FUNCTION_BLOCK "Banda_Poj_+Tryb_Reczny"	// FB 33
//Funkcja realizujaca koncepcje bandy pojedycznej, ktora uwzglednia rowniez tryb 
//reczny. W celu lepszego sterowania trybem recznym nalezy do³o¿yæ:
//-fotokomorki na tyle bandy.
//-fotokomorka na tyle okresla rowniez zajetosc
//-jazda do tylu bandy mozliwa
//-jazda do przodu poza fotokomorke mozliwa gdy nastepna w ruchu i wolna.
//-do³o¿enie okresnia trybu reczny/auto gdzie auto to 1 
//
AUTHOR : Kng
FAMILY : Bandy
NAME : B_dual
VERSION : 0.0
VAR_INPUT
  i_Marka_Bezpieczenstwa : BOOL ;
  i_Rezerwa_1 : BOOL ;	//Zamrozenie stanu pracy
  i_Auto_Reczny : BOOL ;	//1-auto,0-reczny
  i_Foto_Przod : BOOL ;	//Foto na koncu tasmy
  i_Foto_Tyl : BOOL ;	//Foto zapobiegajace wyjechaniu palety do tylu
  i_Zez_Od_Nast : BOOL ;
  i_Paleta_Dost_Od_Nast : BOOL ;
  i_Zez_Reczny_Od_Nast : BOOL ;
  i_Zabierz_Od_Pop : BOOL ;
  i_Zez_Reczny_Od_Pop : BOOL ;
  i_PB_Jazda_Tyl : BOOL ;
  i_PB_Jazda_Przod : BOOL ;
  Czas_Kontroli_Przejazdu : TIME ;
END_VAR
VAR_OUTPUT
  o_Zabierz_Do_Nast : BOOL ;	//Rozkaz pobrania do nast bandy
  o_Zez_Do_Pop : BOOL ;
  o_Paleta_Dost_Do_Pop : BOOL ;
  o_Motor_Lewo : BOOL ;
  o_Motor_Prawo : BOOL ;
  o_Zez_Reczny_Do_Nast : BOOL ;
  o_Zez_Reczny_Do_Pop : BOOL ;
  o_Zajetosc_Nieb : BOOL ;	//Dla bezpieczenstwa transportu
END_VAR
VAR
  Czas_kontrolny : FB 21;
  Help_A_Motor_Lewo : BOOL ;
  S_Help_Zab_Od_Pop : BOOL ;
  Stop_Czas_Kontrolny : BOOL ;
  Zbocze_1 : BOOL ;
  Zbocze_2 : BOOL ;
  Blokada_Wjazdu : BOOL ;
  Help_H_Motor_Prawo : BOOL ;
  Help_H_Motor_Lewo : BOOL ;
  Toggle : BOOL ;	//bit przemienny dla auto i hand
  Help_8 : BOOL ;
  Help_9 : BOOL ;
END_VAR
VAR_TEMP
  Temp_Help_1 : BOOL ;
  Temp_Help_2 : BOOL ;
  Czas_zadany : TIME ;
  Czas_aktualny : TIME ;
END_VAR
BEGIN
NETWORK
TITLE =
//
// B1        B2         foto_1    foto_2         B5        B6
//(\\\\\\\\\\\\\\\\\\)  (\\\\\\\\\\\\\\\\\\)  (\\\\\\\\\\\\\\\\\\)
//                  M1                    M2                     M3
//         
//        zabierz <-- pobierz      |  zabierz    <--  pobierz  
//     zez_do_pop --> zez_od_nast  |  zez_od_pop -->  zez_od_nast
//                                  
//-Uklad dzielony jest na realizowane funkcje
//
//         <----------------------------------------- kierunek
//                  
//
// ten network celowo jest pusty
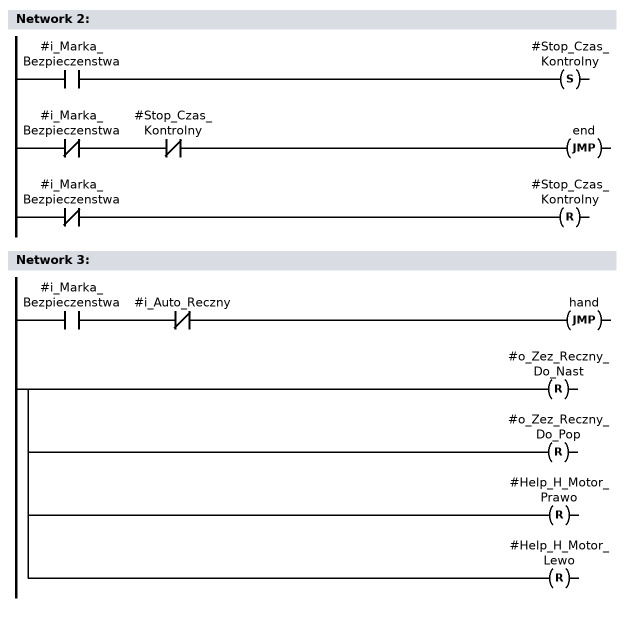
NETWORK
TITLE =
//Sprawdzenie stanu bezpieczenstwa lub freeze
//Skocz jezeli brak marki bezpieczenstwa
//Marka bezpieczenstwa ok gdy wysoki
      A     #i_Marka_Bezpieczenstwa;
      S     #Stop_Czas_Kontrolny;
      AN    #i_Marka_Bezpieczenstwa;
      AN    #Stop_Czas_Kontrolny;
      JC    end;
      AN    #i_Marka_Bezpieczenstwa;
      R     #Stop_Czas_Kontrolny;
NETWORK
TITLE =
//Wyznczenie zbocza pozytywnego i negatywnego
//skok do trybu recznego 
      A     #i_Marka_Bezpieczenstwa;
      AN    #i_Auto_Reczny;
      JC    hand;
//czyszczenie trybu recznego
      SET;
      R     #o_Zez_Reczny_Do_Nast;
      R     #o_Zez_Reczny_Do_Pop;
      R     #Help_H_Motor_Prawo;
      R     #Help_H_Motor_Lewo;
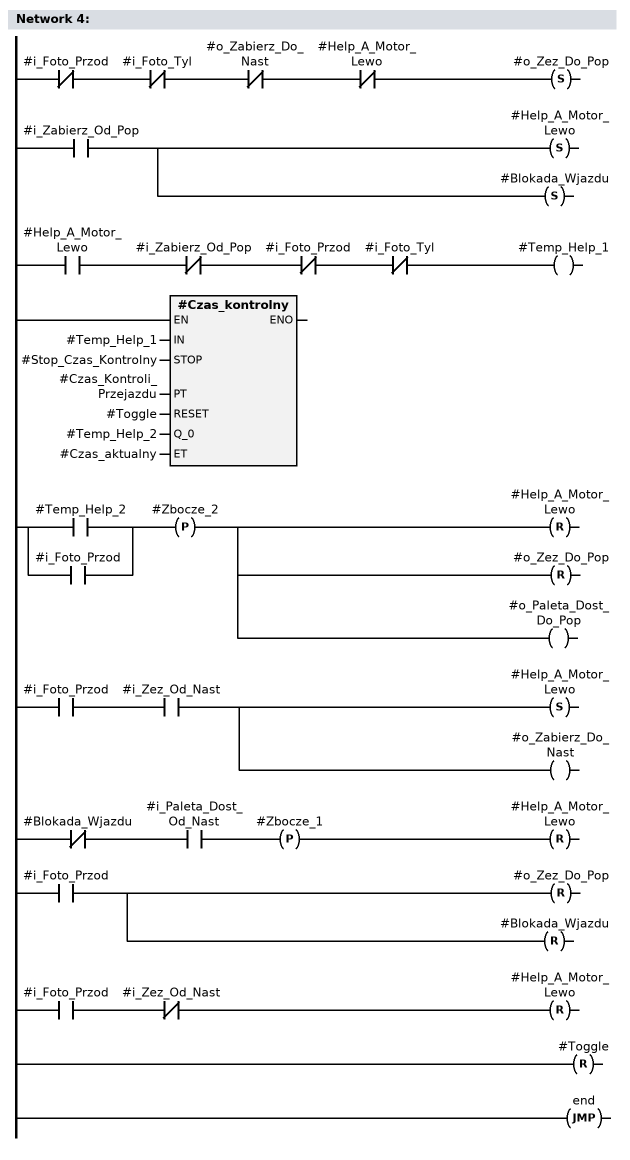
NETWORK
TITLE =
// Opis poszczegolnych krokow i skok do nich
// Tasma poprzednia pusta i bierzaca pusta
      AN    #i_Foto_Przod;
      AN    #i_Foto_Tyl;	//dodano bo hand
      AN    #o_Zabierz_Do_Nast;
      AN    #Help_A_Motor_Lewo;
      S     #o_Zez_Do_Pop;
      A     #i_Zabierz_Od_Pop;
      S     #Help_A_Motor_Lewo;
      S     #Blokada_Wjazdu;
//Warunek gdy pobranie z poprzedniej i miejsce foto srodek
//jest zajete
      A     #Help_A_Motor_Lewo;
      AN    #i_Zabierz_Od_Pop;
      AN    #i_Foto_Przod;
      AN    #i_Foto_Tyl;	//dodano bo hand
      =     #Temp_Help_1;
      CALL  #Czas_kontrolny (
           IN                       := #Temp_Help_1,
           STOP                     := #Stop_Czas_Kontrolny,
           PT                       := #Czas_Kontroli_Przejazdu,
           RESET                    := #Toggle,
           Q_0                      := #Temp_Help_2,
           ET                       := #Czas_aktualny);
//Paleta dostarczona
      A     #Temp_Help_2;
      O;
      A     #i_Foto_Przod;
      FP    #Zbocze_2;
      R     #Help_A_Motor_Lewo;
      R     #o_Zez_Do_Pop;
      =     #o_Paleta_Dost_Do_Pop;
//jest zezwolenie od nastepnej
      A     #i_Foto_Przod;
      A     #i_Zez_Od_Nast;
      S     #Help_A_Motor_Lewo;
      =     #o_Zabierz_Do_Nast;
//Potwierdzenie otrzymania palety
      AN    #Blokada_Wjazdu;
      A     #i_Paleta_Dost_Od_Nast;
      FP    #Zbocze_1;
      R     #Help_A_Motor_Lewo;
//Gdy zajete Foto_1 brak zezwolenia do poprzedniej
      A     #i_Foto_Przod;
      R     #o_Zez_Do_Pop;
      R     #Blokada_Wjazdu;
//warunkowe zakonczenie pracy silnika gdy brak zezwolenia
//z nastepnej
      A     #i_Foto_Przod;
      AN    #i_Zez_Od_Nast;
      R     #Help_A_Motor_Lewo;
//wylacz toggle
      SET;
      R     #Toggle;
//skocz do koniec
      JU    end;
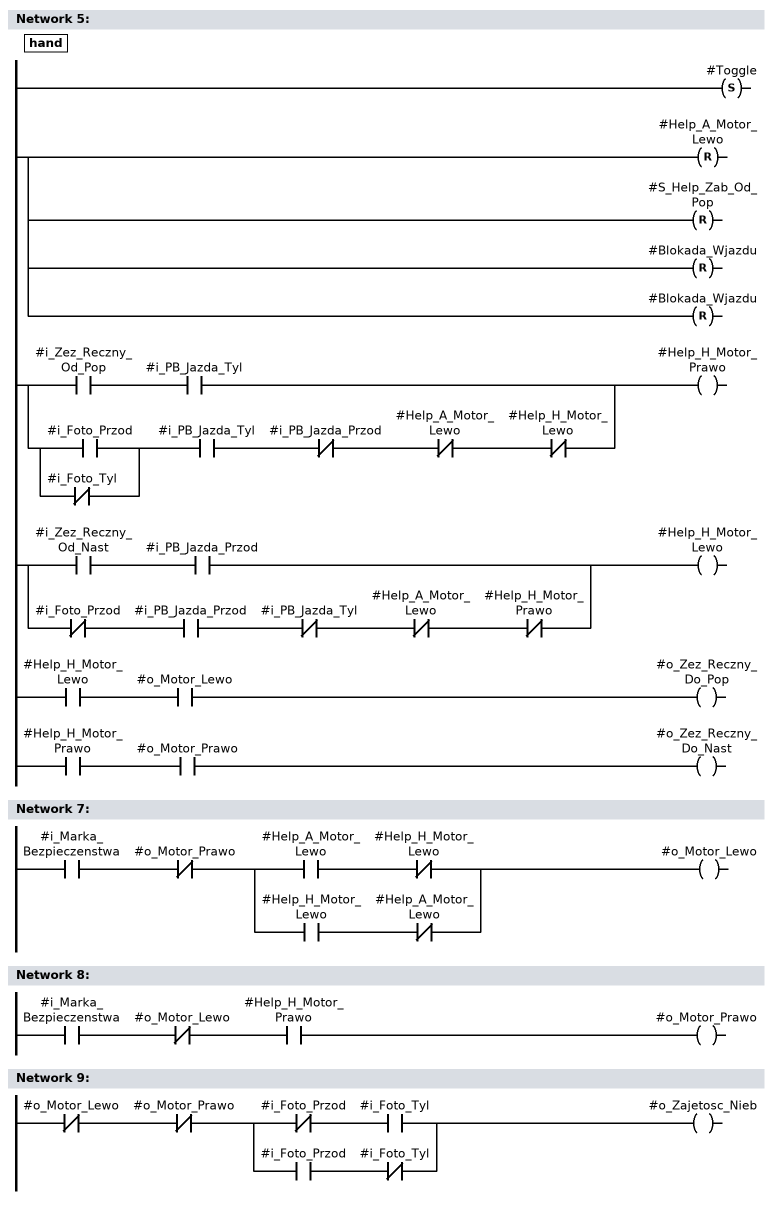
NETWORK
TITLE =
//Tryb reczny
//
hand: NOP   0;
//wlacz toggle
      SET;
      S     #Toggle;
//czyszczenie bitow z automatyki
      SET;
      R     #Help_A_Motor_Lewo;
      R     #S_Help_Zab_Od_Pop;
      R     #Blokada_Wjazdu;
      R     #Blokada_Wjazdu;
//ustawienie przyciskow
//jazda do tylu przycisk tyl
      A     #i_Zez_Reczny_Od_Pop;
      A     #i_PB_Jazda_Tyl;
      O;
      A(;
      O     #i_Foto_Przod;
      ON    #i_Foto_Tyl;
      );
      A(;
      A     #i_PB_Jazda_Tyl;
      AN    #i_PB_Jazda_Przod;
      AN    #Help_A_Motor_Lewo;
      AN    #Help_H_Motor_Lewo;
      );
      =     #Help_H_Motor_Prawo;
//jazda do przodu
      A     #i_Zez_Reczny_Od_Nast;
      A     #i_PB_Jazda_Przod;
      O;
      AN    #i_Foto_Przod;
      A(;
      A     #i_PB_Jazda_Przod;
      AN    #i_PB_Jazda_Tyl;
      AN    #Help_A_Motor_Lewo;
      AN    #Help_H_Motor_Prawo;
      );
      =     #Help_H_Motor_Lewo;
//wystawienie zezwolen do innych band wspolpracujacych recznie
//zezwolenie do tylu 
//zezwolenie do poprzedniej
      A     #Help_H_Motor_Lewo;
      A     #o_Motor_Lewo;
      =     #o_Zez_Reczny_Do_Pop;
//zezwolenie do nastepnej
      A     #Help_H_Motor_Prawo;
      A     #o_Motor_Prawo;
      =     #o_Zez_Reczny_Do_Nast;
NETWORK
TITLE =
//Przypisanie wyjsc
//Koniec skoku
end:  NOP   0;
NETWORK
TITLE =
////jazda automatyka reczny przod
      A     #i_Marka_Bezpieczenstwa;
      AN    #o_Motor_Prawo;
      A(;
      A     #Help_A_Motor_Lewo;
      AN    #Help_H_Motor_Lewo;
      O;
      A     #Help_H_Motor_Lewo;
      AN    #Help_A_Motor_Lewo;
      );
      =     #o_Motor_Lewo;
NETWORK
TITLE =
////Jazda reczny tyl
      A     #i_Marka_Bezpieczenstwa;
      AN    #o_Motor_Lewo;
      A     #Help_H_Motor_Prawo;
      =     #o_Motor_Prawo;
NETWORK
TITLE =
//Zajetosc
      AN    #o_Motor_Lewo;
      AN    #o_Motor_Prawo;
      A(;
      AN    #i_Foto_Przod;
      A     #i_Foto_Tyl;
      O;
      A     #i_Foto_Przod;
      AN    #i_Foto_Tyl;
      );
      =     #o_Zajetosc_Nieb;
NETWORK
TITLE =
//Koniec
//koniec
      BEU;
END_FUNCTION_BLOCK

FUNCTION_BLOCK "Banda_Obr_Bind"	// FB 34
//Program odpowiadajacy za bindowanie produktu na obrotnicy
//
//
AUTHOR : Kng
FAMILY : Bandy
NAME : Band_obr
VERSION : 0.1
VAR_INPUT
  i_Marka_Bezpieczenstwa : BOOL ;
  i_Auto_Reczny : BOOL ;	//gdzie 1-Auto 0 Reczny
  i_Bindownica_Auto : BOOL ;	//Mro¿enie stanu pracy
  i_Foto_Tyl : BOOL ;	//foto poczatek
  i_Foto_Przod : BOOL ;	//foto koniec
  i_Zez_od_Nast : BOOL ;
  i_Zabierz_od_Pop : BOOL ;
  i_Paleta_Dost_Od_Nast : BOOL ;
  i_czuj_0_st_1 : BOOL ;	//0 stopni Wlot/Wylot
  i_czuj_0_st_2 : BOOL ;	//Hamowanie 0 stopni
  i_czuj_90_st_1 : BOOL ;	//Hamowanie 90 stopni
  i_czuj_90_st_2 : BOOL ;	//90 stopni
  i_Czuj_180_st_1 : BOOL ;	//Hamowanie 180 stopni
  i_Czuj_180_st_2 : BOOL ;	//180 stopni
  i_Czuj_270_st_1 : BOOL ;	//Hamowanie 270 stopni
  i_Czuj_270_st_2 : BOOL ;
  i_Bind_Obwod_Ok : BOOL ;	//270 stopni
  i_Bind_Poz_Podst : BOOL ;
  i_Bind_Syg_Got : BOOL ;
  i_Bind_Blad : BOOL ;
  i_Bind_Start_Kon : BOOL ;	//Bindownica start koniec wiazania
  i_PB_Obr_Prawo : BOOL ;
  i_PB_Obr_Lewo : BOOL ;
  i_Zawsze_True : BOOL ;	//Zawsze jeden do pomocy
  i_PB_Jazda_Przod : BOOL ;
  i_PB_Jazda_Tyl : BOOL ;
  i_PB_Cykl_Start : BOOL ;
  i_PB_Cykl_Stop : BOOL ;
  i_Zez_Reczny_Od_Pop : BOOL ;
  i_Zez_Reczny_Od_Nast : BOOL ;
  i_Reset_Krokow : BOOL ;
  i_Reset_Bledow : BOOL ;
  i_Rezerwa_1 : BOOL ;
  i_Rezerwa_2 : BOOL ;
  i_Rezerwa_3 : BOOL ;
  i_Rezerwa_4 : BOOL ;
END_VAR
VAR_OUTPUT
  o_Zez_do_Pop : BOOL ;
  o_Paleta_Dost_Do_Pop : BOOL ;
  o_Zabierz_do_Nast : BOOL ;
  o_Motor_1_lewo : BOOL ;
  o_Motor_1_prawo : BOOL ;
  o_Motor_1_Wolno : BOOL ;
  o_Motor_2_obr_s_Lewo : BOOL ;	//Motor obrotnicy,kierunek strona wejscia,szybko
  o_Motor_2_obr_s_Prawo : BOOL ;	//Motor obrotnicy,kierunek strona wyjscia,szybko
  o_Motor_2_Wolno : BOOL ;	//Motor obrotnicy,kierunek strona wejscia,wolno
  o_Bind_Zez_Na_Prace : BOOL ;
  o_Bind_Start_Wiazania : BOOL ;
  o_Bind_Blad_Ogolny : BOOL ;
  o_Zez_Reczny_do_Pop : BOOL ;
  o_Zez_Reczny_do_nast : BOOL ;
  o_Lampka_Bindowanie : BOOL ;
  o_Lampka_Przycisk_Reset : BOOL ;
  o_Blad_Cyklu : BOOL ;
  o_Blad_Ogolny : BOOL ;
  o_Cykl_Bindowania_Trwa : BOOL ;
  o_Rezerwa_2 : BOOL ;
  o_Rezerwa_3 : BOOL ;
END_VAR
VAR
  Sterowanie_Obrotu : FB 54;
  Pozycj_Obr : FB 55;
  Bindowanie : FB 35;
  Pozycjonowanie_Palety : FB 58;
  Kontrola_Rolki_Wlot : FB 20;
  Dojazd_Rolki_Wlot : FB 20;
  Opuszczenie_Bandy : FB 20;	//Czas kontrolny wjazdu palety
  Tim_Rezerwa_1 : FB 20;
  Tim_Rezerwa_2 : FB 20;
  Tim_Rezerwa_3 : SFB 4;	//Timer opozniajacy bindowanie
  Silniki_nie_pracuja : BOOL ;
  Help_A_Motor_1_lewo : BOOL ;
  Help_A_Motor_1_prawo : BOOL ;
  Help_A_Motor_1_wolno : BOOL ;
  Help_H_Motor_1_lewo : BOOL ;
  Help_H_Motor_1_prawo : BOOL ;
  Help_H_Motor_1_Wolno : BOOL ;
  Help_Motor_2_obr_lewo : BOOL ;
  Help_Motor_2_obr_prawo : BOOL ;
  Help_Motor_2_Wolno : BOOL ;
  Help_AP_Motor_1_Lewo : BOOL ;
  Help_AP_Motor_1_Prawo : BOOL ;
  Help_AP_Motor_1_Wolno : BOOL ;
  Pobranie_Wlot : BOOL ;
  Filtr_Rolki_Wlot : BOOL ;
  Stop_Czas_Kontrolny : BOOL ;
  H1_Doj_Rolki_Wlot : BOOL ;
  H2_Doj_Rolki_Wlot : BOOL ;
  Oddanie_Palety : BOOL ;
  Zbocze_1 : BOOL ;
  Toggle : BOOL ;	//Sygnal zamienny auto reczny
  Paleta_rowno_na_stan : BOOL ;
  Help_B_Zez_Na_Prace : BOOL ;
  Help_B_Start_Wiazan : BOOL ;
  Help_B_Blad_Ogolny : BOOL ;
  Help_Bin_Koniec_Cyklu : BOOL ;
  H_Start_Cyklu_Bind_Auto : BOOL ;
  H_Reset_Cyklu_Bind : BOOL ;
  H_Auto_Reczny : BOOL ;
  Auto_Reczny_W : BOOL ;
  Silnik_Rolek_Nie_Pracuje : BOOL ;
  Reset_Konca_Cyklu : BOOL ;
  Zbocze_2 : BOOL ;
  Help_PB_Start : BOOL ;
  H_Silnik_Rolek_Pracuje : BOOL ;
  H_Zez_do_Pop : BOOL ;
  H_Zabierz_do_Nast : BOOL ;
  H_Cykl_Bind_Trwa : BOOL ;
  Zbocze_3 : BOOL ;
  H_Blad_Cyklu : BOOL ;
  H_Marka_Bezp_Obr : BOOL ;
  H_Marka_Bezp_Poz : BOOL ;
  H_Auto_Reczny_Ster_Obr : BOOL ;
  H_Start_Cyklu_Bind_Recz : BOOL ;
  H_Reset_Srodka : BOOL ;	//Reset paleta na srodku
  H2_Start_Cyklu_Bind_Recz : BOOL ;
  H46 : BOOL ;
  H49 : BOOL ;
  H50 : BOOL ;
  Help_Cykl_Start_Reczny : BOOL ;
  H52 : BOOL ;
  H54 : BOOL ;
  H55 : BOOL ;
  H56 : BOOL ;
  H57 : BOOL ;
  H58 : INT ;
  H59 : BOOL ;
  H60 : BOOL ;	//Pozycja talerza osiagnieta
  H62 : BOOL ;
  H61 : INT ;
  H63 : BOOL ;
  H64 : BOOL ;
  H65 : BOOL ;
  H66 : BOOL ;
  H67 : BOOL ;
  H68 : BOOL ;
  H69 : BOOL ;
  H70 : BOOL ;
  H72 : BOOL ;
  H40 : BOOL ;
  H38 : BOOL ;
  H37 : BOOL ;
  H36 : BOOL ;
  H35 : BOOL ;
  H34 : BOOL ;
  H33 : BOOL ;
  H32 : BOOL ;
  H31 : BOOL ;
  H30 : BOOL ;
  H29 : BOOL ;
  H28 : BOOL ;	//Pozycjonowanie palety
  H27 : BOOL ;
  H26 : BOOL ;
END_VAR
VAR_TEMP
  Temp_Help_1 : BOOL ;
  Temp_Help_2 : BOOL ;
  Czas_zadany : TIME ;
  Czas_aktualny : TIME ;
  Czas_Kontroli_Przejazdu : TIME ;
  Czas_Monitora_Najazdu : TIME ;
  Czas_Opoznienia_Bind : TIME ;
END_VAR
BEGIN
NETWORK
TITLE =
//                   
//Wlot                                Wylot
//()()()()|()()()()|  ()()()  |()()()()|()()()()
//()()()()|()()()()| ()()()() |()()()()|()()()()
//()()()()|()()()()| ()()()() |()()()()|()()()()
//()()()()|()()()()| ()()()() |()()()()|()()()()
//()()()()|()()()()|  ()()()  |()()()()|()()()()
//
//      
//         
//          pobierz --> zabierz   |     pobierz --> zabierz   
//     zez_od_nast <-- zez_do_pop | zez_od_nast <-- zez_od_pop
//                                  
//-Uklad dzielony jest na realizowane funkcje
//
//         
//                  
//
// ten network celowo jest pusty
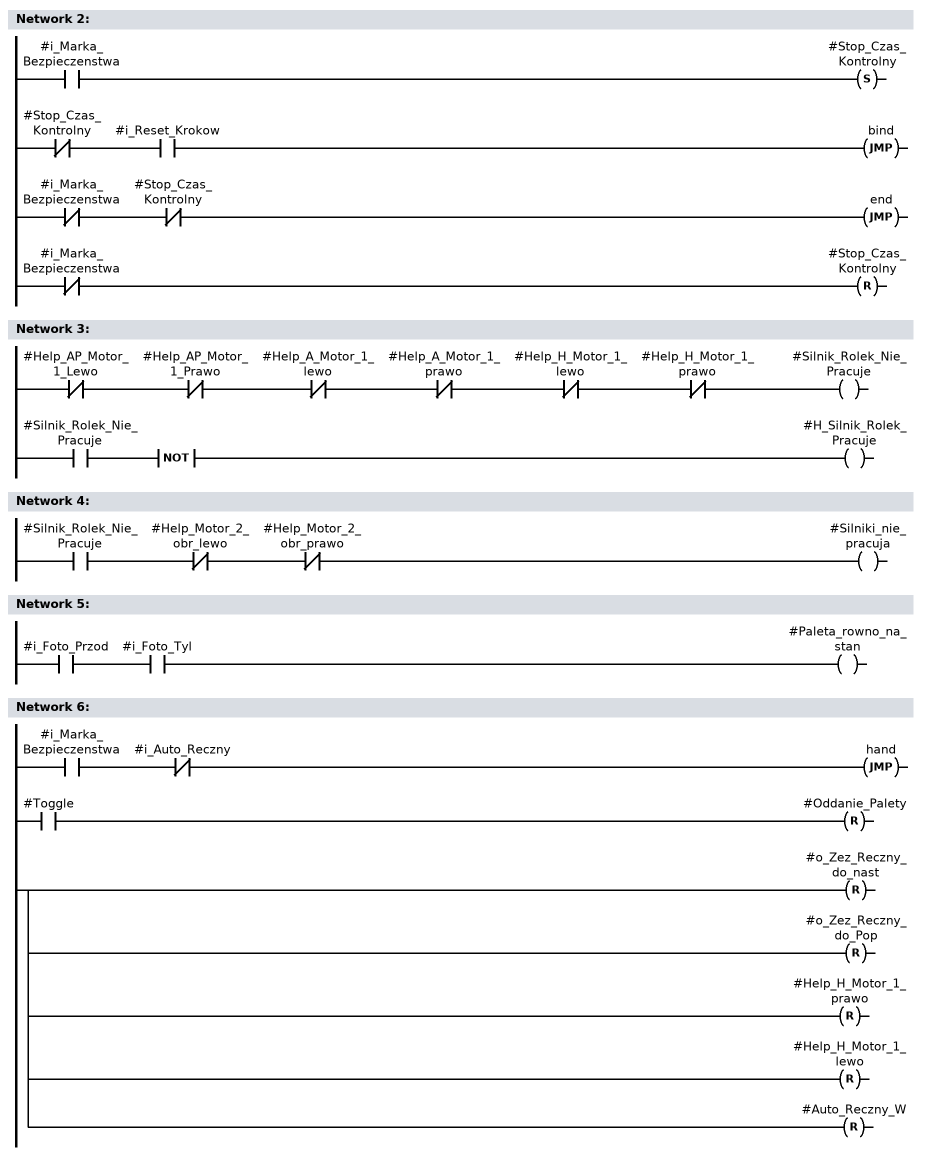
NETWORK
TITLE =
//Wyznczenie zbocza pozytywnego i negatywnego
//Skocz jezeli brak marki bezpieczenstwa
//Marka bezpieczenstwa ok gdy wysoki
//Freeze ok gdy niski
      A     #i_Marka_Bezpieczenstwa;
      S     #Stop_Czas_Kontrolny;
//skocz aby zrobic reset podczas stopu
      AN    #Stop_Czas_Kontrolny;
      A     #i_Reset_Krokow;
      JC    bind;
      AN    #i_Marka_Bezpieczenstwa;
      AN    #Stop_Czas_Kontrolny;
      JC    end;
      AN    #i_Marka_Bezpieczenstwa;
      R     #Stop_Czas_Kontrolny;
NETWORK
TITLE =
//Sprawdzenie czy rolki nie pracuja 
      AN    #Help_AP_Motor_1_Lewo;
      AN    #Help_AP_Motor_1_Prawo;
      AN    #Help_A_Motor_1_lewo;
      AN    #Help_A_Motor_1_prawo;
      AN    #Help_H_Motor_1_lewo;
      AN    #Help_H_Motor_1_prawo;
      =     #Silnik_Rolek_Nie_Pracuje;
      A     #Silnik_Rolek_Nie_Pracuje;
      NOT;
      =     #H_Silnik_Rolek_Pracuje;
NETWORK
TITLE =
//Silniki nie pracuja
//
      A     #Silnik_Rolek_Nie_Pracuje;
      AN    #Help_Motor_2_obr_lewo;
      AN    #Help_Motor_2_obr_prawo;
      =     #Silniki_nie_pracuja;
NETWORK
TITLE =
//Sprawdzenie czy paleta lezy na stanowisku
//sprawdzenie czy paleta lezy OK
      A     #i_Foto_Przod;
      A     #i_Foto_Tyl;
      =     #Paleta_rowno_na_stan;
NETWORK
TITLE =
//Skok do trybu recznego 
//skok do trybu recznego 
      A     #i_Marka_Bezpieczenstwa;
      AN    #i_Auto_Reczny;
      JC    hand;
//Powrot z trybu recznego do auto
      A     #Toggle;
      R     #Oddanie_Palety;
//czyszczenie trybu recznego
      SET;
      R     #o_Zez_Reczny_do_nast;
      R     #o_Zez_Reczny_do_Pop;
      R     #Help_H_Motor_1_prawo;
      R     #Help_H_Motor_1_lewo;
      R     #Auto_Reczny_W;
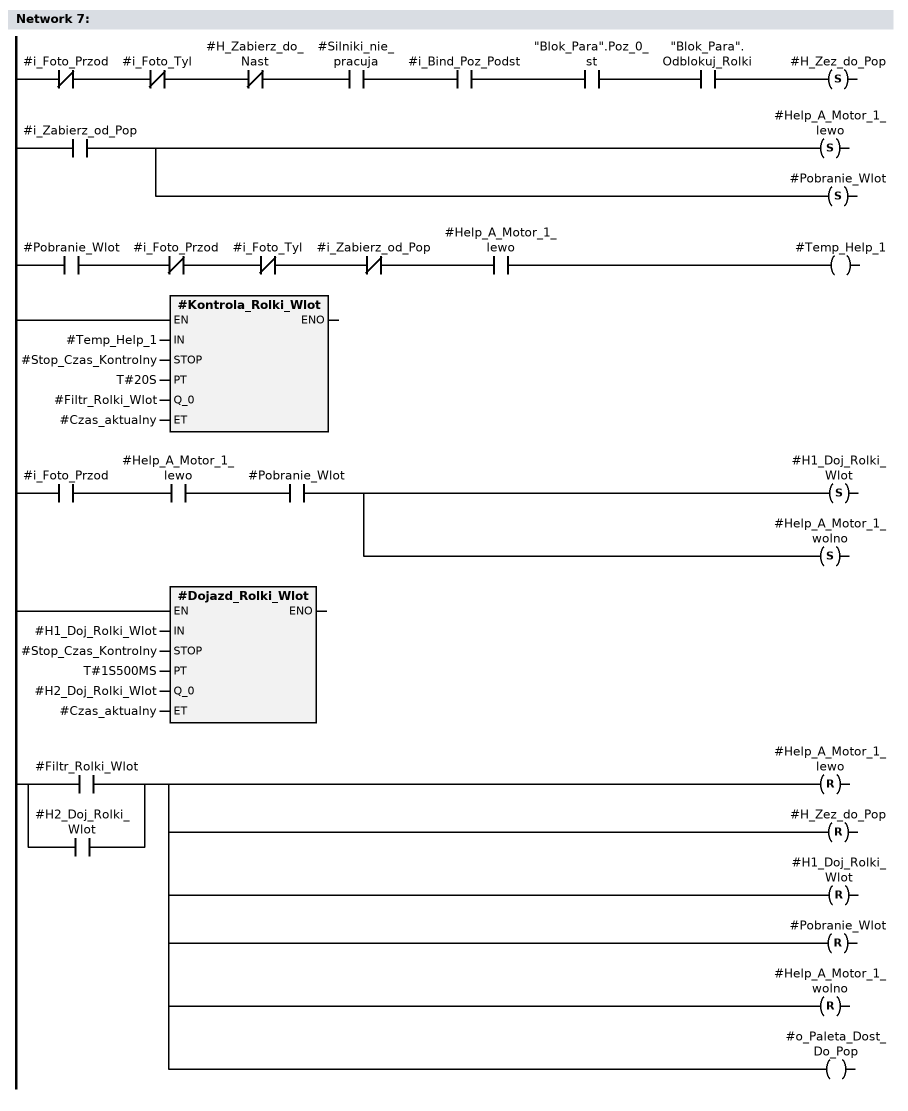
NETWORK
TITLE =
//Wjazd palety na stanowisko bindowania
// Opis poszczegolnych krokow i skok do nich
// Tasma poprzednia pusta i bierzaca pusta
      AN    #i_Foto_Przod;
      AN    #i_Foto_Tyl;
      AN    #H_Zabierz_do_Nast;
      A     #Silniki_nie_pracuja;
      A     #i_Bind_Poz_Podst;
      A     "Blok_Para".Poz_0_st;
      A     "Blok_Para".Odblokuj_Rolki;
      S     #H_Zez_do_Pop;
//gdy sygnal zabierzto blokada wjazdu
      A     #i_Zabierz_od_Pop;
      S     #Help_A_Motor_1_lewo;
      S     #Pobranie_Wlot;
//Czas kontrolny wjazdu na bande
      A     #Pobranie_Wlot;
      AN    #i_Foto_Przod;
      AN    #i_Foto_Tyl;
      AN    #i_Zabierz_od_Pop;
      A     #Help_A_Motor_1_lewo;
      =     #Temp_Help_1;
//Czas kontrolny dojazdu na stanowisko pracy
      CALL  #Kontrola_Rolki_Wlot (
           IN                       := #Temp_Help_1,
           STOP                     := #Stop_Czas_Kontrolny,
           PT                       := T#20S,
           Q_0                      := #Filtr_Rolki_Wlot,
           ET                       := #Czas_aktualny);
//Dojazd na pozycje na obrotnicy
      A     #i_Foto_Przod;
      A     #Help_A_Motor_1_lewo;
      A     #Pobranie_Wlot;
      S     #H1_Doj_Rolki_Wlot;
      S     #Help_A_Motor_1_wolno;
      CALL  #Dojazd_Rolki_Wlot (
           IN                       := #H1_Doj_Rolki_Wlot,
           STOP                     := #Stop_Czas_Kontrolny,
           PT                       := T#1S500MS,
           Q_0                      := #H2_Doj_Rolki_Wlot,
           ET                       := #Czas_aktualny);
//Koniec pobierania palety z wlotu 1
      A     #Filtr_Rolki_Wlot;
      O;
      A     #H2_Doj_Rolki_Wlot;
      R     #Help_A_Motor_1_lewo;
      R     #H_Zez_do_Pop;
      R     #H1_Doj_Rolki_Wlot;
      R     #Pobranie_Wlot;
      R     #Help_A_Motor_1_wolno;
      =     #o_Paleta_Dost_Do_Pop;
//-------------------------------------------------
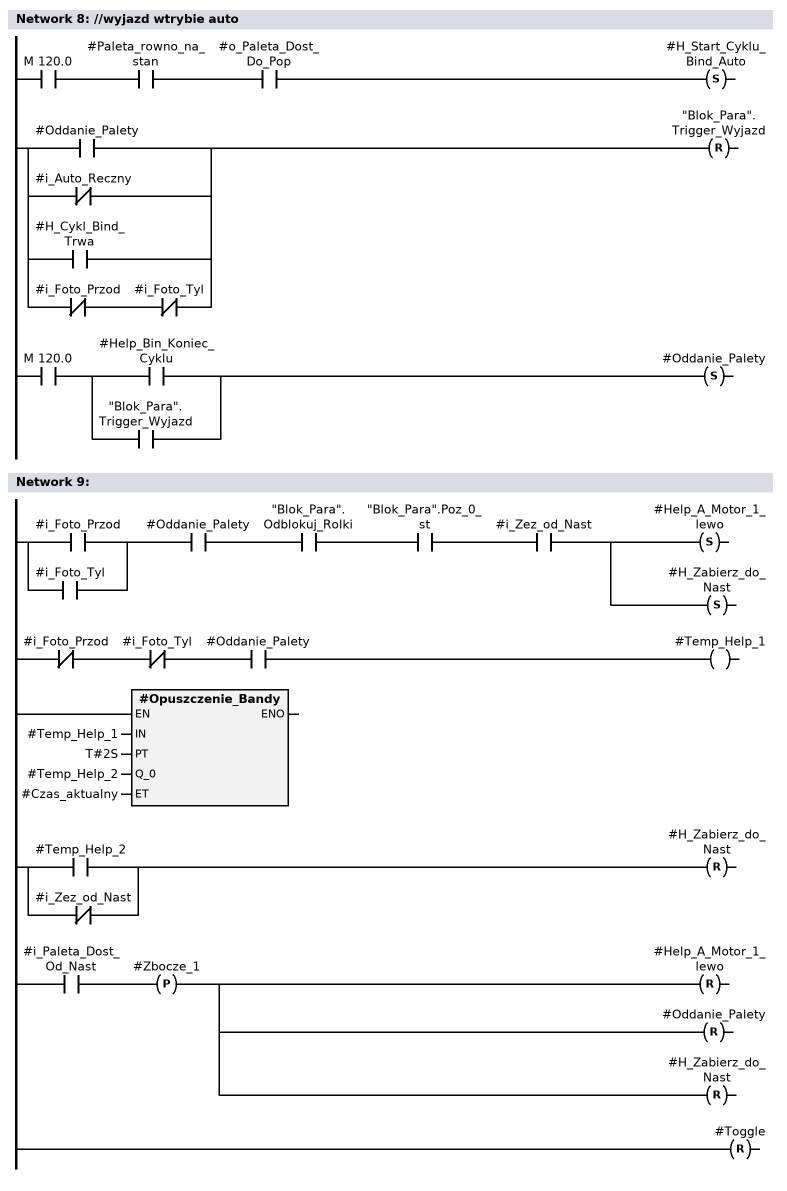
NETWORK
TITLE = //wyjazd wtrybie auto
//Bindowanie
//rozpoczecie cyklu bindowania
      A     M 120.0;
      A     #Paleta_rowno_na_stan;
      A     #o_Paleta_Dost_Do_Pop;
      S     #H_Start_Cyklu_Bind_Auto;
//zakolnczenie cyku bindowania
      O     #Oddanie_Palety;
      ON    #i_Auto_Reczny;
      O     #H_Cykl_Bind_Trwa;
      O(;
      AN    #i_Foto_Przod;
      AN    #i_Foto_Tyl;
      );
      R     "Blok_Para".Trigger_Wyjazd;
      A     M 120.0;
      A(;
      O     #Help_Bin_Koniec_Cyklu;
      O     "Blok_Para".Trigger_Wyjazd;
      );
      S     #Oddanie_Palety;
NETWORK
TITLE =
//Wyjazd palety z bindowania
//jest zezwolenie od nastepnej
//Oczekiwanie na zezwolenie
      O     #i_Foto_Przod;
      O     #i_Foto_Tyl;
      A     #Oddanie_Palety;
      A     "Blok_Para".Odblokuj_Rolki;
      A     "Blok_Para".Poz_0_st;
      A     #i_Zez_od_Nast;
      S     #Help_A_Motor_1_lewo;
      S     #H_Zabierz_do_Nast;
//reset sygn³u zabierz
      AN    #i_Foto_Przod;
      AN    #i_Foto_Tyl;
      A     #Oddanie_Palety;
      =     #Temp_Help_1;
      CALL  #Opuszczenie_Bandy (
           IN                       := #Temp_Help_1,
           PT                       := T#2S,
           Q_0                      := #Temp_Help_2,
           ET                       := #Czas_aktualny);
      A     #Temp_Help_2;
      O;
      AN    #i_Zez_od_Nast;
      R     #H_Zabierz_do_Nast;
      A     #i_Paleta_Dost_Od_Nast;
      FP    #Zbocze_1;
      R     #Help_A_Motor_1_lewo;
      R     #Oddanie_Palety;
      R     #H_Zabierz_do_Nast;
      SET;
//wylacz toggle
      R     #Toggle;
//skocz do koniec
NETWORK
TITLE =
//Resetowanie Startu bindowania gdy bindowanie zalaczone
con:  NOP   0;
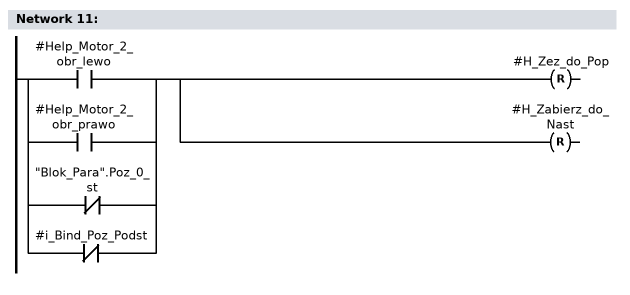
NETWORK
TITLE =
//Wrunkowe resetowanie zezwolen
// warunkowy reset zezwolenia
      O     #Help_Motor_2_obr_lewo;
      O     #Help_Motor_2_obr_prawo;
      ON    "Blok_Para".Poz_0_st;
      ON    #i_Bind_Poz_Podst;
      R     #H_Zez_do_Pop;
      R     #H_Zabierz_do_Nast;
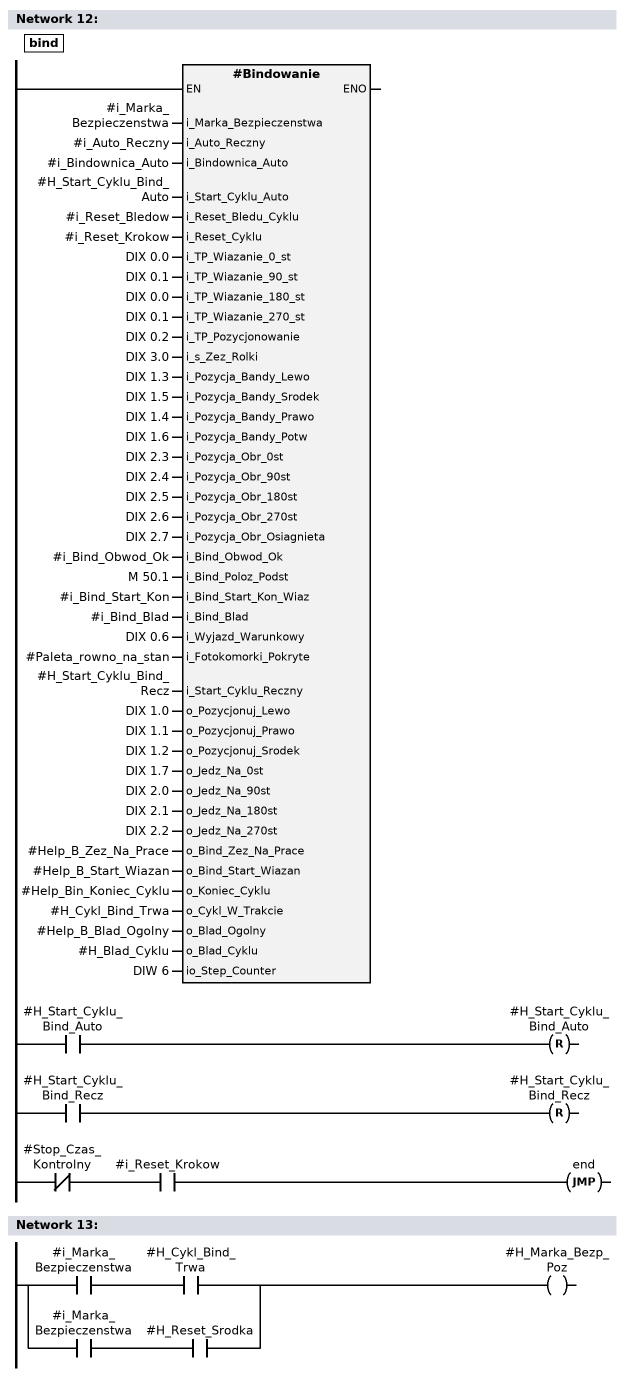
NETWORK
TITLE =
//Bindownica
bind: NOP   0;
      CALL  #Bindowanie (
           i_Marka_Bezpieczenstwa   := #i_Marka_Bezpieczenstwa,
           i_Auto_Reczny            := #i_Auto_Reczny,
           i_Bindownica_Auto        := #i_Bindownica_Auto,
           i_Start_Cyklu_Auto       := #H_Start_Cyklu_Bind_Auto,
           i_Reset_Bledu_Cyklu      := #i_Reset_Bledow,
           i_Reset_Cyklu            := #i_Reset_Krokow,
           i_TP_Wiazanie_0_st       := DIX 0.0,
           i_TP_Wiazanie_90_st      := DIX 0.1,
           i_TP_Wiazanie_180_st     := DIX 0.0,
           i_TP_Wiazanie_270_st     := DIX 0.1,
           i_TP_Pozycjonowanie      := DIX 0.2,
           i_s_Zez_Rolki            := DIX 3.0,
           i_Pozycja_Bandy_Lewo     := DIX 1.3,
           i_Pozycja_Bandy_Srodek   := DIX 1.5,
           i_Pozycja_Bandy_Prawo    := DIX 1.4,
           i_Pozycja_Bandy_Potw     := DIX 1.6,
           i_Pozycja_Obr_0st        := DIX 2.3,
           i_Pozycja_Obr_90st       := DIX 2.4,
           i_Pozycja_Obr_180st      := DIX 2.5,
           i_Pozycja_Obr_270st      := DIX 2.6,
           i_Pozycja_Obr_Osiagnieta := DIX 2.7,
           i_Bind_Obwod_Ok          := #i_Bind_Obwod_Ok,
           i_Bind_Poloz_Podst       := M 50.1,
           i_Bind_Start_Kon_Wiaz    := #i_Bind_Start_Kon,
           i_Bind_Blad              := #i_Bind_Blad,
           i_Wyjazd_Warunkowy       := DIX 0.6,
           i_Fotokomorki_Pokryte    := #Paleta_rowno_na_stan,
           i_Start_Cyklu_Reczny     := #H_Start_Cyklu_Bind_Recz,
           o_Pozycjonuj_Lewo        := DIX 1.0,
           o_Pozycjonuj_Prawo       := DIX 1.1,
           o_Pozycjonuj_Srodek      := DIX 1.2,
           o_Jedz_Na_0st            := DIX 1.7,
           o_Jedz_Na_90st           := DIX 2.0,
           o_Jedz_Na_180st          := DIX 2.1,
           o_Jedz_Na_270st          := DIX 2.2,
           o_Bind_Zez_Na_Prace      := #Help_B_Zez_Na_Prace,
           o_Bind_Start_Wiazan      := #Help_B_Start_Wiazan,
           o_Koniec_Cyklu           := #Help_Bin_Koniec_Cyklu,
           o_Cykl_W_Trakcie         := #H_Cykl_Bind_Trwa,
           o_Blad_Ogolny            := #Help_B_Blad_Ogolny,
           o_Blad_Cyklu             := #H_Blad_Cyklu,
           io_Step_Counter          := DIW 6);
      A     #H_Start_Cyklu_Bind_Auto;
      R     #H_Start_Cyklu_Bind_Auto;
      A     #H_Start_Cyklu_Bind_Recz;
      R     #H_Start_Cyklu_Bind_Recz;
      AN    #Stop_Czas_Kontrolny;
      A     #i_Reset_Krokow;
      JC    end;
//Resetowanie warunkowe marki cyklu startu 
//Powrot do ominiecia 
NETWORK
TITLE =
//Marka bepieczenstwa Pozycjononwanie
      A     #i_Marka_Bezpieczenstwa;
      A     #H_Cykl_Bind_Trwa;
      O;
      A     #i_Marka_Bezpieczenstwa;
      A     #H_Reset_Srodka;
      =     #H_Marka_Bezp_Poz;
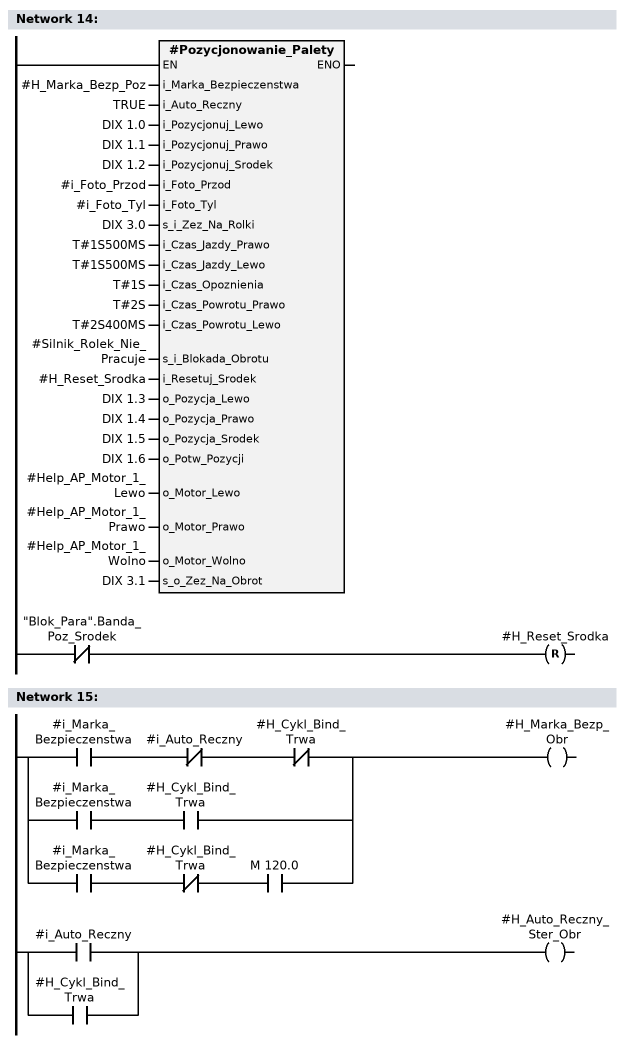
NETWORK
TITLE =
//Pozycjonowanie palety
      CALL  #Pozycjonowanie_Palety (
           i_Marka_Bezpieczenstwa   := #H_Marka_Bezp_Poz,
           i_Auto_Reczny            := TRUE,
           i_Pozycjonuj_Lewo        := DIX 1.0,
           i_Pozycjonuj_Prawo       := DIX 1.1,
           i_Pozycjonuj_Srodek      := DIX 1.2,
           i_Foto_Przod             := #i_Foto_Przod,
           i_Foto_Tyl               := #i_Foto_Tyl,
           s_i_Zez_Na_Rolki         := DIX 3.0,
           i_Czas_Jazdy_Prawo       := T#1S500MS,
           i_Czas_Jazdy_Lewo        := T#1S500MS,
           i_Czas_Opoznienia        := T#1S,
           i_Czas_Powrotu_Prawo     := T#2S,
           i_Czas_Powrotu_Lewo      := T#2S400MS,
           s_i_Blokada_Obrotu       := #Silnik_Rolek_Nie_Pracuje,
           i_Resetuj_Srodek         := #H_Reset_Srodka,
           o_Pozycja_Lewo           := DIX 1.3,
           o_Pozycja_Prawo          := DIX 1.4,
           o_Pozycja_Srodek         := DIX 1.5,
           o_Potw_Pozycji           := DIX 1.6,
           o_Motor_Lewo             := #Help_AP_Motor_1_Lewo,
           o_Motor_Prawo            := #Help_AP_Motor_1_Prawo,
           o_Motor_Wolno            := #Help_AP_Motor_1_Wolno,
           s_o_Zez_Na_Obrot         := DIX 3.1);	//czas pozycjonowania prawo / czas pozycjonowania lewo / czas powrotu od prwej / czas powrotu od lewej
      AN    "Blok_Para".Banda_Poz_Srodek;
      R     #H_Reset_Srodka;
NETWORK
TITLE =
//Marka bezpieczenstwa sterowania obrotu
      A     #i_Marka_Bezpieczenstwa;
      AN    #i_Auto_Reczny;
      AN    #H_Cykl_Bind_Trwa;
      O;
      A     #i_Marka_Bezpieczenstwa;
      A     #H_Cykl_Bind_Trwa;
      O;
      A     #i_Marka_Bezpieczenstwa;
      AN    #H_Cykl_Bind_Trwa;
      A     M 120.0;
      =     #H_Marka_Bezp_Obr;
      A     #i_Auto_Reczny;
      O;
      A     #H_Cykl_Bind_Trwa;
      =     #H_Auto_Reczny_Ster_Obr;
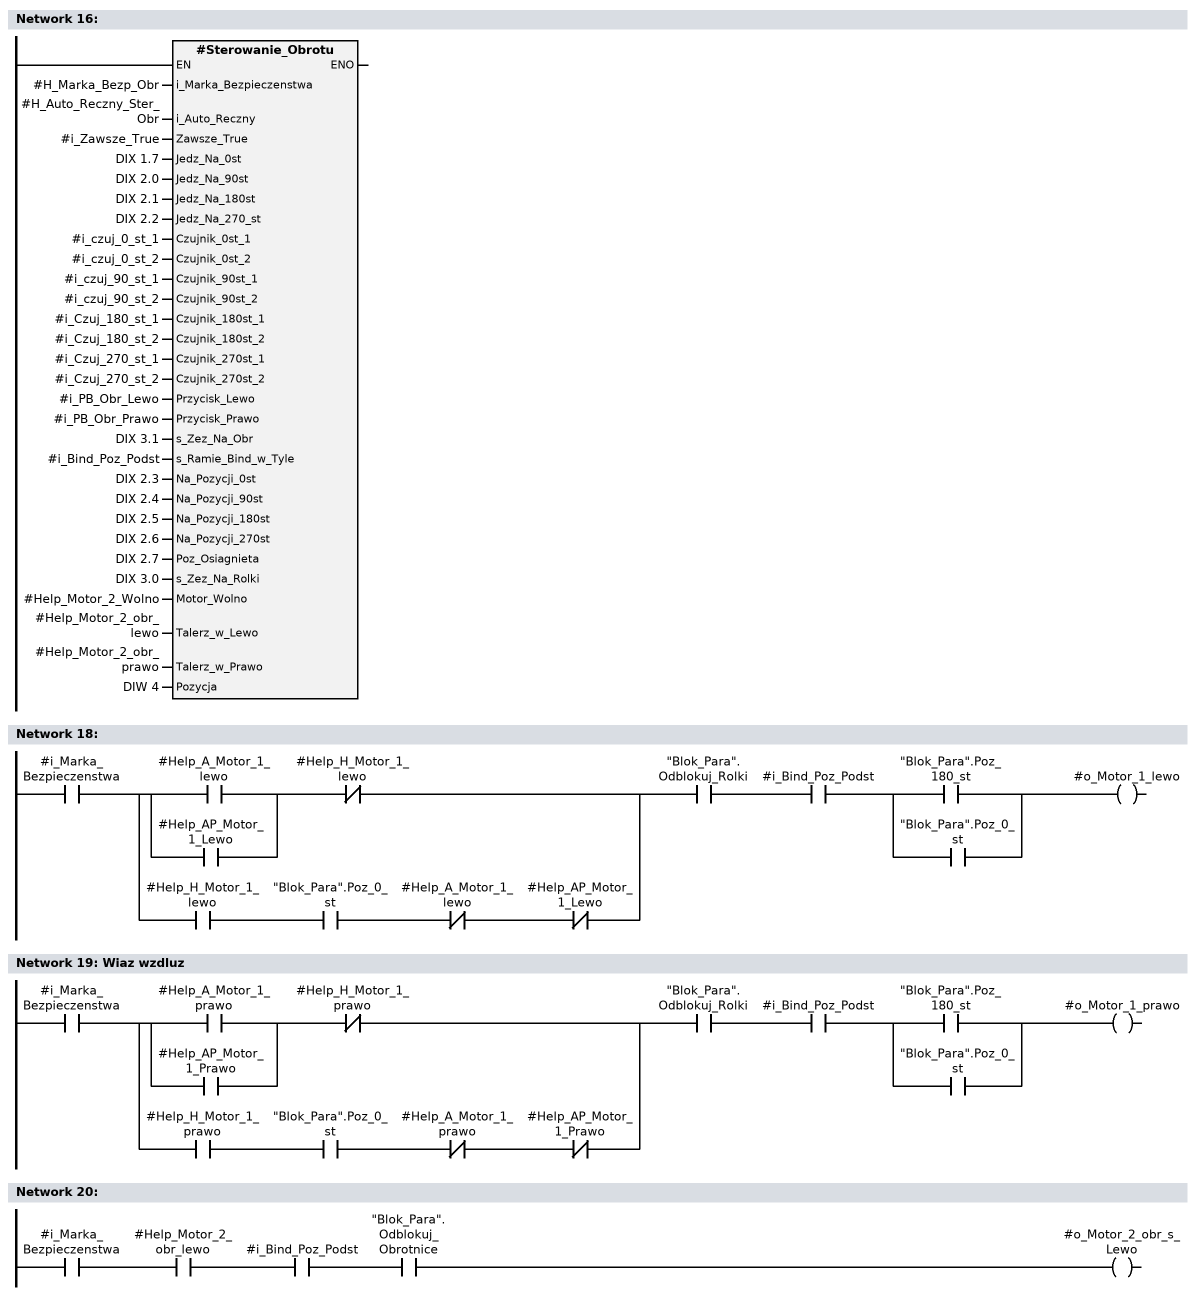
NETWORK
TITLE =
//Obrot na pozycje 
      CALL  #Sterowanie_Obrotu (
           i_Marka_Bezpieczenstwa   := #H_Marka_Bezp_Obr,
           i_Auto_Reczny            := #H_Auto_Reczny_Ster_Obr,
           Zawsze_True              := #i_Zawsze_True,
           Jedz_Na_0st              := DIX 1.7,
           Jedz_Na_90st             := DIX 2.0,
           Jedz_Na_180st            := DIX 2.1,
           Jedz_Na_270_st           := DIX 2.2,
           Czujnik_0st_1            := #i_czuj_0_st_1,
           Czujnik_0st_2            := #i_czuj_0_st_2,
           Czujnik_90st_1           := #i_czuj_90_st_1,
           Czujnik_90st_2           := #i_czuj_90_st_2,
           Czujnik_180st_1          := #i_Czuj_180_st_1,
           Czujnik_180st_2          := #i_Czuj_180_st_2,
           Czujnik_270st_1          := #i_Czuj_270_st_1,
           Czujnik_270st_2          := #i_Czuj_270_st_2,
           Przycisk_Lewo            := #i_PB_Obr_Lewo,
           Przycisk_Prawo           := #i_PB_Obr_Prawo,
           s_Zez_Na_Obr             := DIX 3.1,
           s_Ramie_Bind_w_Tyle      := #i_Bind_Poz_Podst,
           Na_Pozycji_0st           := DIX 2.3,
           Na_Pozycji_90st          := DIX 2.4,
           Na_Pozycji_180st         := DIX 2.5,
           Na_Pozycji_270st         := DIX 2.6,
           Poz_Osiagnieta           := DIX 2.7,
           s_Zez_Na_Rolki           := DIX 3.0,
           Motor_Wolno              := #Help_Motor_2_Wolno,
           Talerz_w_Lewo            := #Help_Motor_2_obr_lewo,
           Talerz_w_Prawo           := #Help_Motor_2_obr_prawo,
           Pozycja                  := DIW 4);
NETWORK
TITLE =
//Wyzwalanie wyjsc
end:  NOP   0;
NETWORK
TITLE =
//Motor rolki lewo
      A     #i_Marka_Bezpieczenstwa;
      A(;
      A(;
      O     #Help_A_Motor_1_lewo;
      O     #Help_AP_Motor_1_Lewo;
      );
      AN    #Help_H_Motor_1_lewo;
      O;
      A     #Help_H_Motor_1_lewo;
      A     "Blok_Para".Poz_0_st;
      AN    #Help_A_Motor_1_lewo;
      AN    #Help_AP_Motor_1_Lewo;
      );
      A     "Blok_Para".Odblokuj_Rolki;
      A     #i_Bind_Poz_Podst;
      A(;
      O     "Blok_Para".Poz_180_st;
      O     "Blok_Para".Poz_0_st;
      );
      =     #o_Motor_1_lewo;
NETWORK
TITLE = Wiaz wzdluz
//Motor rolki prawo
      A     #i_Marka_Bezpieczenstwa;
      A(;
      A(;
      O     #Help_A_Motor_1_prawo;
      O     #Help_AP_Motor_1_Prawo;
      );
      AN    #Help_H_Motor_1_prawo;
      O;
      A     #Help_H_Motor_1_prawo;
      A     "Blok_Para".Poz_0_st;
      AN    #Help_A_Motor_1_prawo;
      AN    #Help_AP_Motor_1_Prawo;
      );
      A     "Blok_Para".Odblokuj_Rolki;
      A     #i_Bind_Poz_Podst;
      A(;
      O     "Blok_Para".Poz_180_st;
      O     "Blok_Para".Poz_0_st;
      );
      =     #o_Motor_1_prawo;
NETWORK
TITLE =
//motor obrotnica lewo
      A     #i_Marka_Bezpieczenstwa;
      A     #Help_Motor_2_obr_lewo;
      A     #i_Bind_Poz_Podst;
      A     "Blok_Para".Odblokuj_Obrotnice;
      =     #o_Motor_2_obr_s_Lewo;
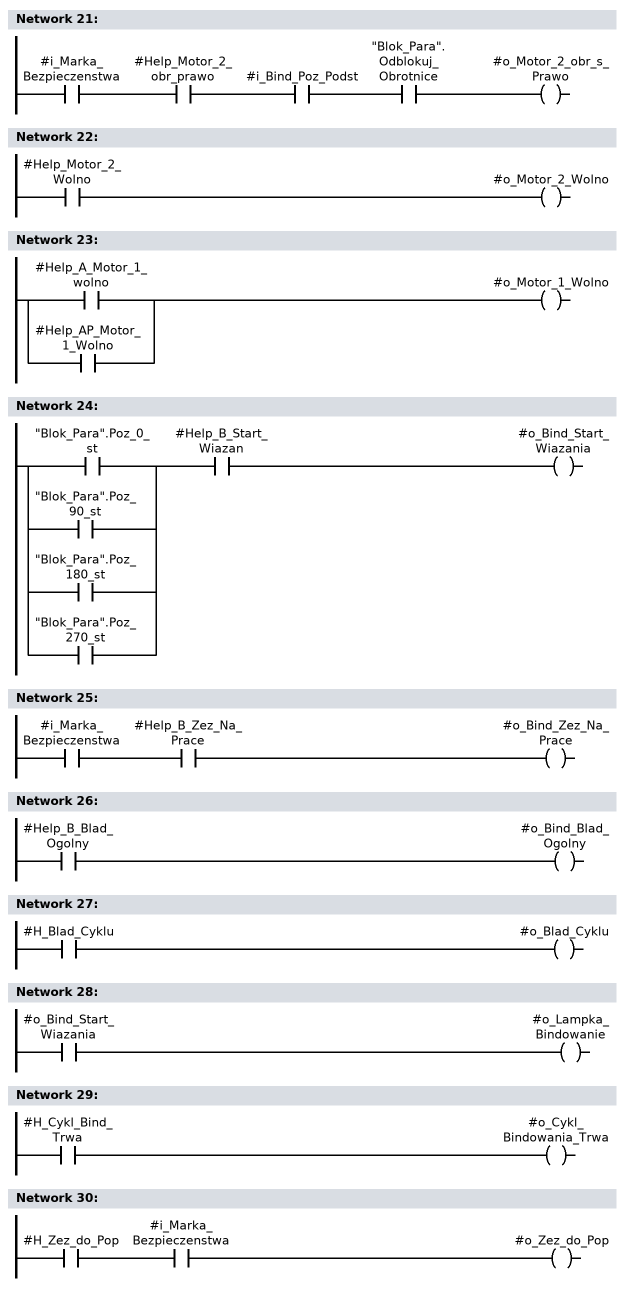
NETWORK
TITLE =
//motor obrotnica prawo
      A     #i_Marka_Bezpieczenstwa;
      A     #Help_Motor_2_obr_prawo;
      A     #i_Bind_Poz_Podst;
      A     "Blok_Para".Odblokuj_Obrotnice;
      =     #o_Motor_2_obr_s_Prawo;
NETWORK
TITLE =
//motor obrotnica wolno
      A     #Help_Motor_2_Wolno;
      =     #o_Motor_2_Wolno;
NETWORK
TITLE =
//Motor rolki wolno
      O     #Help_A_Motor_1_wolno;
      O     #Help_AP_Motor_1_Wolno;
      =     #o_Motor_1_Wolno;
NETWORK
TITLE =
//zalaczeni wiazarki. Uwaga ze wzgledu na gasnacy sygnal
//      A     #i_Marka_Bezpieczenstwa
      A(;
      O     "Blok_Para".Poz_0_st;
      O     "Blok_Para".Poz_90_st;
      O     "Blok_Para".Poz_180_st;
      O     "Blok_Para".Poz_270_st;
      );
      A     #Help_B_Start_Wiazan;
      =     #o_Bind_Start_Wiazania;
NETWORK
TITLE =
//Zezwolenie na prace bindownicy
      A     #i_Marka_Bezpieczenstwa;
      A     #Help_B_Zez_Na_Prace;
      =     #o_Bind_Zez_Na_Prace;
NETWORK
TITLE =
//Blad ogolny Bindownicy
      A     #Help_B_Blad_Ogolny;
      =     #o_Bind_Blad_Ogolny;
NETWORK
TITLE =
//Blad Cyklu
      A     #H_Blad_Cyklu;
      =     #o_Blad_Cyklu;
NETWORK
TITLE =
//Lampka bindowanie
      A     #o_Bind_Start_Wiazania;
      =     #o_Lampka_Bindowanie;
NETWORK
TITLE =
//Cykl bindowanie trwa
      A     #H_Cykl_Bind_Trwa;
      =     #o_Cykl_Bindowania_Trwa;
NETWORK
TITLE =
//Zezwolenie do poprzedniej 
      A     #H_Zez_do_Pop;
      A     #i_Marka_Bezpieczenstwa;
      =     #o_Zez_do_Pop;
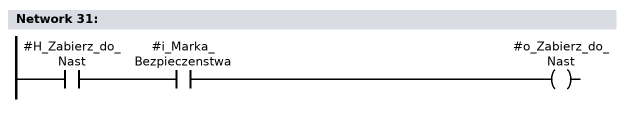
NETWORK
TITLE =
//Zabierz do nast
      A     #H_Zabierz_do_Nast;
      A     #i_Marka_Bezpieczenstwa;
      =     #o_Zabierz_do_Nast;
NETWORK
TITLE =
//Zakonczenie dzialania programu
//
//zakonczenie programu
      BEU;
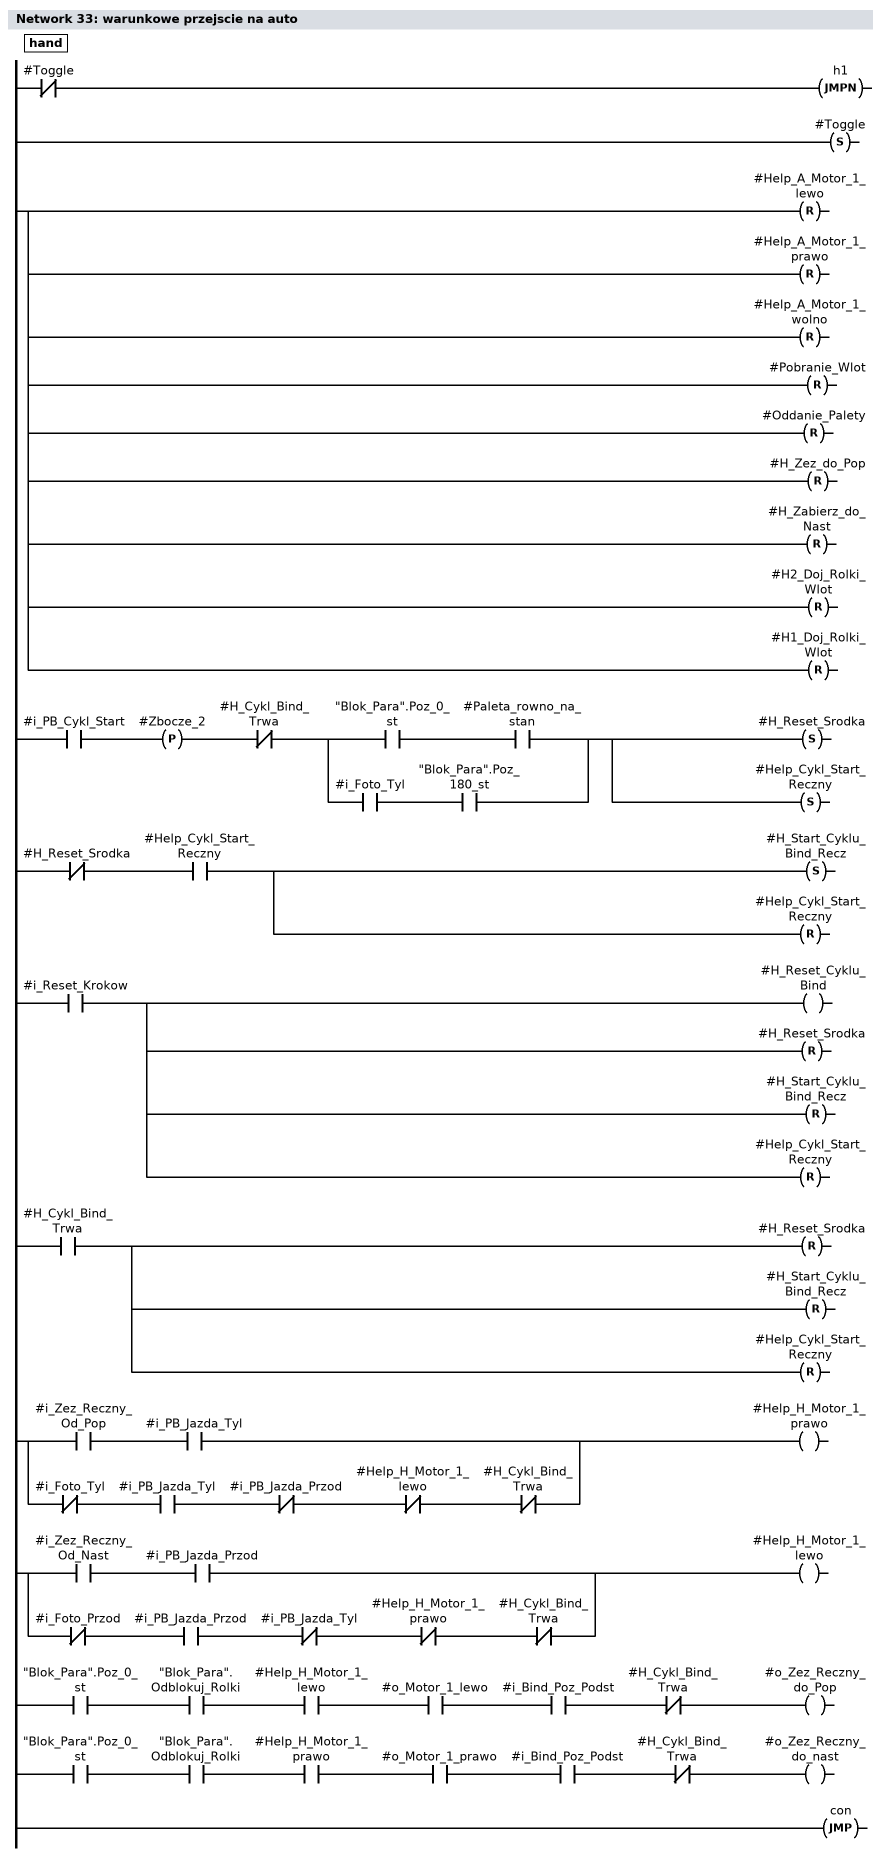
NETWORK
TITLE = warunkowe przejscie na auto
//Tryb jazdy banda rolkowa po zalaczeniu recznego. Po wejsciu w tryb reczny 
//jezeli 
//sie nic nie robilo to mozna wyjsc i maszyna pracuje dalej. 
//***********************Tryb Rezczny*************************
//************************************************************
hand: NOP   0;
//************************************************
//Pierwsze wejscie to resetuj
      AN    #Toggle;
      JCN   h1;
//tu wpisac kod toggle
h1:   NOP   0;
//*************************************************
//wlacz toggle
      SET;
      S     #Toggle;
//**************************************************
//czyszczenie bitow z automatyki
      SET;
      R     #Help_A_Motor_1_lewo;
      R     #Help_A_Motor_1_prawo;
      R     #Help_A_Motor_1_wolno;
      R     #Pobranie_Wlot;
      R     #Oddanie_Palety;
      R     #H_Zez_do_Pop;
      R     #H_Zabierz_do_Nast;
      R     #H2_Doj_Rolki_Wlot;
      R     #H1_Doj_Rolki_Wlot;
//***************************************************
//Start automatyki w trybie recznym
      A     #i_PB_Cykl_Start;
      FP    #Zbocze_2;
      AN    #H_Cykl_Bind_Trwa;
      A(;
      O(;
      A     "Blok_Para".Poz_0_st;
      A     #Paleta_rowno_na_stan;
      );
      O(;
      A     #i_Foto_Tyl;
      A     "Blok_Para".Poz_180_st;
      );
      );
      S     #H_Reset_Srodka;
      S     #Help_Cykl_Start_Reczny;
      AN    #H_Reset_Srodka;
      A     #Help_Cykl_Start_Reczny;
      S     #H_Start_Cyklu_Bind_Recz;
      R     #Help_Cykl_Start_Reczny;
//jezeli start nie dziala to reset wyrownanie fotkomorek
      A     #i_Reset_Krokow;
      =     #H_Reset_Cyklu_Bind;
      R     #H_Reset_Srodka;
      R     #H_Start_Cyklu_Bind_Recz;
      R     #Help_Cykl_Start_Reczny;
//-
      A     #H_Cykl_Bind_Trwa;
      R     #H_Reset_Srodka;
      R     #H_Start_Cyklu_Bind_Recz;
      R     #Help_Cykl_Start_Reczny;
//********************Jazda Reczna*********************
//ustawienie przyciskow
//jazda do tylu przycisk tyl
      A     #i_Zez_Reczny_Od_Pop;
      A     #i_PB_Jazda_Tyl;
      O;
      AN    #i_Foto_Tyl;
      A(;
      A     #i_PB_Jazda_Tyl;
      AN    #i_PB_Jazda_Przod;
      AN    #Help_H_Motor_1_lewo;
      );
      AN    #H_Cykl_Bind_Trwa;
      =     #Help_H_Motor_1_prawo;
//jazda do przodu
      A     #i_Zez_Reczny_Od_Nast;
      A     #i_PB_Jazda_Przod;
      O;
      AN    #i_Foto_Przod;
      A(;
      A     #i_PB_Jazda_Przod;
      AN    #i_PB_Jazda_Tyl;
      AN    #Help_H_Motor_1_prawo;
      );
      AN    #H_Cykl_Bind_Trwa;
      =     #Help_H_Motor_1_lewo;
//wystawienie zezwolen do innych band wspolpracujacych recznie
//zezwolenie do tylu 
//zezwolenie do poprzedniej
      A     "Blok_Para".Poz_0_st;
      A     "Blok_Para".Odblokuj_Rolki;
      A     #Help_H_Motor_1_lewo;
      A     #o_Motor_1_lewo;
      A     #i_Bind_Poz_Podst;
      AN    #H_Cykl_Bind_Trwa;
      =     #o_Zez_Reczny_do_Pop;
//zezwolenie do nastepnej
      A     "Blok_Para".Poz_0_st;
      A     "Blok_Para".Odblokuj_Rolki;
      A     #Help_H_Motor_1_prawo;
      A     #o_Motor_1_prawo;
      A     #i_Bind_Poz_Podst;
      AN    #H_Cykl_Bind_Trwa;
      =     #o_Zez_Reczny_do_nast;
//skok do dalszej czesc programu
      JU    con;
END_FUNCTION_BLOCK

FUNCTION_BLOCK "Blok_Pracy_Bindownicy"	// FB 35
//Funkcja odpowiada za sterowanie calym procesem bindowania
//Jezeli dane zostaly zmienione w trakcie trwania cyklu to dopiero w czasie 
//nowego 
//cyklu zostana przyjete.
//
//
//
VERSION : 0.1
VAR_INPUT
  i_Marka_Bezpieczenstwa : BOOL ;
  i_Auto_Reczny : BOOL ;
  i_Bindownica_Auto : BOOL ;
  i_Start_Cyklu_Auto : BOOL ;
  i_Reset_Bledu_Cyklu : BOOL ;
  i_Reset_Cyklu : BOOL ;	//Sprowadza funkcje do poczatku
  i_Pozycjonuj_Palete : BOOL ;
  i_TP_Wiazanie_0_st : BOOL ;
  i_TP_Wiazanie_90_st : BOOL ;
  i_TP_Wiazanie_180_st : BOOL ;
  i_TP_Wiazanie_270_st : BOOL ;
  i_TP_Pozycjonowanie : BOOL ;
  i_s_Zez_Rolki : BOOL ;
  i_Pozycja_Bandy_Lewo : BOOL ;
  i_Pozycja_Bandy_Srodek : BOOL ;
  i_Pozycja_Bandy_Prawo : BOOL ;
  i_Pozycja_Bandy_Potw : BOOL ;
  i_Pozycja_Obr_0st : BOOL ;
  i_Pozycja_Obr_90st : BOOL ;
  i_Pozycja_Obr_180st : BOOL ;
  i_Pozycja_Obr_270st : BOOL ;
  i_Pozycja_Obr_Osiagnieta : BOOL ;
  i_Bind_Obwod_Ok : BOOL ;
  i_Bind_Poloz_Podst : BOOL ;
  i_Bind_Start_Kon_Wiaz : BOOL ;
  i_Bind_Blad : BOOL ;
  i_Wyjazd_Warunkowy : BOOL ;
  i_Fotokomorki_Pokryte : BOOL ;
  i_Start_Cyklu_Reczny : BOOL ;
  i_Rezerwa_4 : BOOL ;
  i_Rezerwa_5 : BOOL ;
END_VAR
VAR_OUTPUT
  o_Pozycjonuj_Lewo : BOOL ;
  o_Pozycjonuj_Prawo : BOOL ;
  o_Pozycjonuj_Srodek : BOOL ;
  o_Jedz_Na_0st : BOOL ;
  o_Jedz_Na_90st : BOOL ;
  o_Jedz_Na_180st : BOOL ;
  o_Jedz_Na_270st : BOOL ;
  o_Bind_Zez_Na_Prace : BOOL ;
  o_Bind_Start_Wiazan : BOOL ;
  o_Koniec_Cyklu : BOOL ;
  o_Cykl_W_Trakcie : BOOL ;	//informacja ze maszyna jest w trakcie cyklu
  o_Blad_Ogolny : BOOL ;
  o_Blad_Cyklu : BOOL ;
  o_Rezerwa_1 : BOOL ;
  o_Rezerwa_2 : BOOL ;
  o_Rezerwa_3 : BOOL ;
  o_Rezerwa_4 : BOOL ;
END_VAR
VAR_IN_OUT
  io_Step_Counter : INT ;
END_VAR
VAR
  Kontrola_Tranzycji : FB 20;	//Timmer kontrolujacy czy krok jest konczony
  Timer_Pauzy : FB 20;
  Timer_Kon_Strzalu : FB 20;	//Timer kontroli strzalu
  Tim_Rezerwa_2 : FB 20;
  Tim_Rezerwa_3 : FB 20;
  H_Czas_Kontrolny : TIME ;
  Stop_Czas_Kontrolny : BOOL ;
  H_Czas_Pauzy : TIME ;
  Start_Bindowania : BOOL ;
  H_Obr_Na_Poz_X : BOOL ;
  H_Pozycjonuj_Srodek : BOOL ;
  H_Pozycjonuj_Lewo : BOOL ;
  H_Pozycjonuj_Prawo : BOOL ;
  H_Wykonaj_Wiazanie : BOOL ;
  H_Wiazanie_Zak_Pom : BOOL ;
  H_Jedz_Na_Poz_X : BOOL ;
  H_Paleta_Na_Prawo : BOOL ;
  H_Paleta_Na_Srodku : BOOL ;
  H_Paleta_Na_Lewo : BOOL ;
  H_Wiazanie_0_st : BOOL ;
  H_Wiazanie_90_st : BOOL ;
  H_Wiazanie_180_st : BOOL ;
  H_Wiazanie_270_st : BOOL ;
  H_Pozycjonowanie : BOOL ;
  H_Blad : BOOL ;
  Bit_Tranzycji : BOOL ;
  Zbocze_1 : BOOL ;
  H_Bit_Pauzy : BOOL ;
  H_Poczatek_Pauzy : BOOL ;
  H_Koniec_Pauzy : BOOL ;
  Krok_1 : BOOL ;
  Krok_2 : BOOL ;
  Krok_3 : BOOL ;
  Krok_4 : BOOL ;
  Krok_5 : BOOL ;
  Krok_6 : BOOL ;
  Krok_7 : BOOL ;
  Krok_8 : BOOL ;
  Krok_9 : BOOL ;
  Trwa_Krok_1 : BOOL ;
  Trwa_Krok_2 : BOOL ;
  Trwa_Krok_3 : BOOL ;
  Trwa_Krok_4 : BOOL ;
  Trwa_Krok_5 : BOOL ;
  Trwa_Krok_6 : BOOL ;
  Trwa_Krok_7 : BOOL ;
  Trwa_Krok_8 : BOOL ;
  Trwa_Krok_9 : BOOL ;
  Zadanie_1 : BOOL ;
  Zadanie_2 : BOOL ;
  Zadanie_3 : BOOL ;
  Zadanie_4 : BOOL ;
  Zadanie_5 : BOOL ;
  Zadanie_6 : BOOL ;
  Zadanie_10 : BOOL ;
  H_int : INT ;
  H_Pozycja_0_st_ok : BOOL ;
  H_Pozycja_90_st_ok : BOOL ;
  H_Pozycja_180_st_ok : BOOL ;
  H_Pozycja_270_st_ok : BOOL ;
  Zbocze_2 : BOOL ;
  H_Bindownic_Skon_Wiaz : BOOL ;
  H_Help_Koniec_Wiazan : BOOL ;
  H_20 : BOOL ;
  H_30 : BOOL ;
  H_31 : BOOL ;
  H_32 : BOOL ;
  H_22 : BOOL ;
  H_34 : BOOL ;
  H_45 : BOOL ;
  H_23 : BOOL ;
END_VAR
VAR_TEMP
  Help_Bit_1 : BOOL ;
  Help_Bit_2 : BOOL ;
  Bit_Kontroli_Czasu : BOOL ;
  Czas_Aktualny : TIME ;
  Help_Bit_3 : BOOL ;
END_VAR
BEGIN
NETWORK
TITLE =
//Ten network celow jest wolny
//
NETWORK
TITLE =
//Przygotowanie marki bezpieczenstw
      A     #i_Marka_Bezpieczenstwa;
      S     #Stop_Czas_Kontrolny;
      AN    #i_Marka_Bezpieczenstwa;
      R     #Stop_Czas_Kontrolny;
NETWORK
TITLE =
//Przygotowanie do startu
//
//
//********************************************
//Reset konca cyklu
      L     0;
      L     #io_Step_Counter;
      ==I;
      R     #o_Koniec_Cyklu;
//********************************************
//Rozpoczecie bindowania
      A     #o_Koniec_Cyklu;
      JCN   et_1;
      L     0;
      T     #io_Step_Counter;
et_1: NOP   0;
//********************************************
// Start cyklu bindowania
      A     #i_Auto_Reczny;
      A     #i_Start_Cyklu_Auto;
      AN    #o_Cykl_W_Trakcie;
      O;
      A     #i_Start_Cyklu_Reczny;
      AN    #i_Auto_Reczny;
      AN    #o_Cykl_W_Trakcie;
      S     #Start_Bindowania;
//********************************************
//Zresetowanie bitow startowych
      A     #i_Auto_Reczny;
      A     #Start_Bindowania;
      JCN   et_a;
      L     2;
      T     #io_Step_Counter;
      SET;
      R     #Start_Bindowania;
et_a: NOP   0;
      AN    #i_Auto_Reczny;
      A     #Start_Bindowania;
      JCN   et_r;
      L     1;
      T     #io_Step_Counter;
      SET;
      R     #Start_Bindowania;
et_r: NOP   0;
//********************************************
//Gdy reset wcisniety to kasuj wszystkie bity
      AN    #i_Auto_Reczny;
      A     #i_Reset_Cyklu;
      JCN   et_3;
      L     0;
      T     #io_Step_Counter;
      SET;
      R     #o_Koniec_Cyklu;
      R     #o_Cykl_W_Trakcie;
      JU    clrs;
et_3: NOP   0;
//********************************************
//Pozycjonowanie palety
      A     #i_Pozycjonuj_Palete;
      JCN   et_4;
      L     10;
      T     #io_Step_Counter;
et_4: NOP   0;
//********************************************
//Maszyna w trakcie cyklu bindowania
      L     #io_Step_Counter;
      L     0;
      <>I;
      =     #o_Cykl_W_Trakcie;
//********************************************
//Przypisanie jazdy do nowych pozycji gdy koniec cyklu
      A     #o_Cykl_W_Trakcie;
      JC    et_5;
//0st
      A     #i_TP_Wiazanie_0_st;
      =     #H_Wiazanie_0_st;
//90st
      A     #i_TP_Wiazanie_90_st;
      =     #H_Wiazanie_90_st;
//180st
      A     #i_TP_Wiazanie_180_st;
      =     #H_Wiazanie_180_st;
//270st
      A     #i_TP_Wiazanie_270_st;
      =     #H_Wiazanie_270_st;
//Pozycjonowanie
      A     #i_TP_Pozycjonowanie;
      =     #H_Pozycjonowanie;
et_5: NOP   0;
//********************************************
//Wyjazd warunkowy
      A     #i_Pozycja_Obr_0st;
      A     #i_Auto_Reczny;
      A     #i_Wyjazd_Warunkowy;
      AN    #o_Cykl_W_Trakcie;
      JCN   et_6;
      L     6;
      T     #io_Step_Counter;
et_6: NOP   0;
NETWORK
TITLE =
//Lista Zadan Pracy
//
//**************Zadania  ***********************
//Srodkowanie dla 0 
      L     #io_Step_Counter;
      L     1;
      ==I;
      =     #Zadanie_1;
//0st
      L     #io_Step_Counter;
      L     2;
      ==I;
      =     #Zadanie_2;
//90st
      L     #io_Step_Counter;
      L     3;
      ==I;
      =     #Zadanie_3;
//180st
      L     #io_Step_Counter;
      L     4;
      ==I;
      =     #Zadanie_4;
//270st
      L     #io_Step_Counter;
      L     5;
      ==I;
      =     #Zadanie_5;
//powrot 0st
      L     #io_Step_Counter;
      L     6;
      ==I;
      =     #Zadanie_6;
//reset
      L     #io_Step_Counter;
      L     10;
      ==I;
      =     #Zadanie_10;
NETWORK
TITLE =
//Maszyna z krokiem nr 0
//Jezeli wartosc licznika 0 to
//Wyczysc wszystko i wyjdz
      L     #io_Step_Counter;
      L     0;
      ==I;
      JC    clrs;
NETWORK
TITLE =
      A     #Zadanie_1;
      JCN   u_1;
      SET;
      S     #Krok_1;
//***************************************************
//Krok 1 - jedz na pozycje 0st 
      A     #Krok_1;
      AN    #Krok_2;
      R     #H_Paleta_Na_Srodku;
      A     #Krok_1;
      A(;
      O     #i_Pozycja_Obr_0st;
      O     #i_Pozycja_Obr_180st;
      );
      S     #Krok_2;
//****************************************************
//jezeli nie ma pozycji to wyzeruj
      AN    #Krok_2;
      JC    zer;
//****************************************************
//Krok 2 - Jezeli tryb z pozycjonowaniem to wysrodkuj palete
      A     #H_Paleta_Na_Srodku;
      AN    #Krok_3;
      S     #Krok_3;
      R     #H_Pozycjonuj_Srodek;
      R     #H_Paleta_Na_Srodku;
//-
      A     #Krok_2;
      AN    #Krok_3;
      =     #Trwa_Krok_2;
      S     #H_Pozycjonuj_Srodek;
      JC    res;
//Krok 3 - Przejscie do kroku inkrementu
      A     #Krok_3;
      S     #Krok_7;
//Krok 7 - Zadanie ukonczone przejdz do nastepnego zadania
      A     #Krok_7;
      JC    inc;
u_1:  NOP   0;
NETWORK
TITLE =
//Zadanie nr 2 wiazanie na pozycji 0st
//**************Zadanie 2 ***********************
      A     #Zadanie_2;
      JCN   u_2;
//***************************************************
//Wyskocz jezeli brak wiazania dla 0st
      AN    #H_Wiazanie_0_st;
      JC    inc;
//***************************************************
//Rozpoczecie grafu
      SET;
      S     #Krok_1;
//***************************************************
//Krok 1 - jedz na pozycje 0st 
      A     #H_Obr_Na_Poz_X;
      S     #Krok_2;
      R     #H_Obr_Na_Poz_X;
      R     #H_Jedz_Na_Poz_X;
//-
      A     #Krok_1;
      AN    #Krok_2;
      =     #Trwa_Krok_1;
      S     #H_Jedz_Na_Poz_X;
      JC    j_1;
//***************************************************
//Krok 2 - Jezeli tryb z pozycjonowaniem to wyœrodkuj palete
      A     #H_Pozycjonowanie;
      A     #H_Paleta_Na_Srodku;
      AN    #Krok_3;
      O;
      AN    #H_Pozycjonowanie;
      AN    #Krok_3;
      S     #Krok_3;
      R     #H_Pozycjonuj_Srodek;
      R     #H_Paleta_Na_Srodku;
//-
      A     #Krok_2;
      AN    #Krok_3;
      =     #Trwa_Krok_2;
      S     #H_Pozycjonuj_Srodek;
      JC    res;
//***************************************************
//Krok 3 - Dla 0 stopni pozycjonuj w prawo przed strza³em
      A     #H_Pozycjonowanie;
      A     #H_Paleta_Na_Prawo;
      O;
      AN    #H_Pozycjonowanie;
      S     #Krok_4;
      R     #H_Pozycjonuj_Prawo;
      R     #H_Paleta_Na_Prawo;
//-
      A     #Krok_3;
      AN    #Krok_4;
      =     #Trwa_Krok_3;
      S     #H_Pozycjonuj_Prawo;
      JC    pp;
//***************************************************
//Krok 4 -Wykonaj wiazanie
      A     #H_Wiazanie_Zak_Pom;
      S     #Krok_5;
      R     #H_Wykonaj_Wiazanie;
      R     #H_Wiazanie_Zak_Pom;
      R     #H_Bindownic_Skon_Wiaz;
//-
      A     #Krok_4;
      AN    #Krok_5;
      =     #Trwa_Krok_4;
      S     #H_Wykonaj_Wiazanie;
      JC    bind;
//*****************************************************
//Krok 5 - Przerwa po zwiazaniu
      A     #H_Koniec_Pauzy;
      S     #Krok_6;
      R     #H_Poczatek_Pauzy;
      R     #H_Koniec_Pauzy;
//-
      L     T#2S;
      T     #H_Czas_Pauzy;
//-
      A     #Krok_5;
      AN    #Krok_6;
      =     #Trwa_Krok_5;
      S     #H_Poczatek_Pauzy;
      JC    wait;
//*****************************************************
//Krok 6 - Jezeli tryb z pozycjonowaniem to wyœrodkuj palete
      A     #H_Pozycjonowanie;
      A     #H_Paleta_Na_Srodku;
      AN    #Krok_7;
      O;
      AN    #H_Pozycjonowanie;
      AN    #Krok_7;
      S     #Krok_7;
      R     #H_Pozycjonuj_Srodek;
      R     #H_Paleta_Na_Srodku;
//-
      A     #Krok_6;
      AN    #Krok_7;
      =     #Trwa_Krok_6;
      S     #H_Pozycjonuj_Srodek;
      JC    res;
//***************************************************
//Krok 7 - Zadanie ukonczone przejdz do nastepnego zadania
      A     #Krok_7;
      JC    inc;
u_2:  NOP   0;
NETWORK
TITLE =
//Zadanie nr 3 wiazanie na pozycji 90st
//**************Zadanie 3 ***********************
      A     #Zadanie_3;
      JCN   u_3;
//***************************************************
//Wyskocz jezeli brak wiazania dla 0st
      AN    #H_Wiazanie_90_st;
      JC    inc;
//***************************************************
//Rozpoczecie grafu
      SET;
      S     #Krok_1;
//***************************************************
//Krok 1 - jedz na pozycje 90st 
      A     #H_Obr_Na_Poz_X;
      S     #Krok_2;
      R     #H_Obr_Na_Poz_X;
      R     #H_Jedz_Na_Poz_X;
//-
      A     #Krok_1;
      AN    #Krok_2;
      =     #Trwa_Krok_1;
      S     #H_Jedz_Na_Poz_X;
      JC    j_2;
//***************************************************
//Przejdz pominiete kroki
      A     #Krok_2;
      S     #Krok_3;
//-
      A     #Krok_3;
      S     #Krok_4;
//***************************************************
//Krok 4 -Wykonaj wiazanie
      A     #H_Wiazanie_Zak_Pom;
      S     #Krok_5;
      R     #H_Wykonaj_Wiazanie;
      R     #H_Wiazanie_Zak_Pom;
      R     #H_Bindownic_Skon_Wiaz;
//-
      A     #Krok_4;
      AN    #Krok_5;
      =     #Trwa_Krok_4;
      S     #H_Wykonaj_Wiazanie;
      JC    bind;
//*****************************************************
//Krok 5 - Przerwa po zwiazaniu
      A     #H_Koniec_Pauzy;
      S     #Krok_6;
      R     #H_Poczatek_Pauzy;
      R     #H_Koniec_Pauzy;
//-
      L     T#2S;
      T     #H_Czas_Pauzy;
//-
      A     #Krok_5;
      AN    #Krok_6;
      =     #Trwa_Krok_5;
      S     #H_Poczatek_Pauzy;
      JC    wait;
//*****************************************************
//Krok 6
      A     #Krok_6;
      S     #Krok_7;
//***************************************************
//Krok 7 - Zadanie ukonczone przejdz do nastepnego zadania
      A     #Krok_7;
      JC    inc;
u_3:  NOP   0;
NETWORK
TITLE =
//Zadanie nr 4 wiazanie na pozycji 180st
//**************Zadanie 4 ***********************
      A     #Zadanie_4;
      JCN   u_4;
//***************************************************
//Wyskocz jezeli brak wiazania dla 0st
      AN    #H_Wiazanie_180_st;
      JC    inc;
//***************************************************
//Rozpoczecie grafu
      SET;
      S     #Krok_1;
//***************************************************
//Krok 1 - jedz na pozycje 0st 
      A     #H_Obr_Na_Poz_X;
      S     #Krok_2;
      R     #H_Obr_Na_Poz_X;
      R     #H_Jedz_Na_Poz_X;
//-
      A     #Krok_1;
      AN    #Krok_2;
      =     #Trwa_Krok_1;
      S     #H_Jedz_Na_Poz_X;
      JC    j_3;
//***************************************************
//Krok 2 - Jezeli tryb z pozycjonowaniem to wyœrodkuj palete
      A     #H_Pozycjonowanie;
      A     #H_Paleta_Na_Srodku;
      AN    #Krok_3;
      O;
      AN    #H_Pozycjonowanie;
      AN    #Krok_3;
      S     #Krok_3;
      R     #H_Pozycjonuj_Srodek;
      R     #H_Paleta_Na_Srodku;
//-
      A     #Krok_2;
      AN    #Krok_3;
      =     #Trwa_Krok_2;
      S     #H_Pozycjonuj_Srodek;
      JC    res;
//***************************************************
//Krok 3 - Dla 180 stopni pozycjonuj w lewo przed strza³em
      A     #H_Pozycjonowanie;
      A     #H_Paleta_Na_Lewo;
      O;
      AN    #H_Pozycjonowanie;
      S     #Krok_4;
      R     #H_Pozycjonuj_Lewo;
      R     #H_Paleta_Na_Lewo;
//-
      A     #Krok_3;
      AN    #Krok_4;
      =     #Trwa_Krok_3;
      S     #H_Pozycjonuj_Lewo;
      JC    pl;
//***************************************************
//Krok 4 -Wykonaj wiazanie
      A     #H_Wiazanie_Zak_Pom;
      S     #Krok_5;
      R     #H_Wykonaj_Wiazanie;
      R     #H_Wiazanie_Zak_Pom;
      R     #H_Bindownic_Skon_Wiaz;
//-
      A     #Krok_4;
      AN    #Krok_5;
      =     #Trwa_Krok_4;
      S     #H_Wykonaj_Wiazanie;
      JC    bind;
//*****************************************************
//Krok 5 - Przerwa po zwiazaniu
      A     #H_Koniec_Pauzy;
      S     #Krok_6;
      R     #H_Poczatek_Pauzy;
      R     #H_Koniec_Pauzy;
//-
      L     T#2S;
      T     #H_Czas_Pauzy;
//-
      A     #Krok_5;
      AN    #Krok_6;
      =     #Trwa_Krok_5;
      S     #H_Poczatek_Pauzy;
      JC    wait;
//*****************************************************
//Krok 6 - Jezeli tryb z pozycjonowaniem to wyœrodkuj palete
      A     #H_Pozycjonowanie;
      A     #H_Paleta_Na_Srodku;
      AN    #Krok_7;
      O;
      AN    #H_Pozycjonowanie;
      AN    #Krok_7;
      S     #Krok_7;
      R     #H_Pozycjonuj_Srodek;
      R     #H_Paleta_Na_Srodku;
//-
      A     #Krok_6;
      AN    #Krok_7;
      =     #Trwa_Krok_6;
      S     #H_Pozycjonuj_Srodek;
      JC    res;
//***************************************************
//Krok 7 - Zadanie ukonczone przejdz do nastepnego zadania
      A     #Krok_7;
      JC    inc;
u_4:  NOP   0;
NETWORK
TITLE =
//Zadanie nr 3 wiazanie na pozycji 270st
//**************Zadanie 5 ***********************
      A     #Zadanie_5;
      JCN   u_5;
//***************************************************
//Wyskocz jezeli brak wiazania dla 0st
      AN    #H_Wiazanie_270_st;
      JC    inc;
//***************************************************
//Rozpoczecie grafu
      SET;
      S     #Krok_1;
//***************************************************
//Krok 1 - jedz na pozycje 90st 
      A     #H_Obr_Na_Poz_X;
      S     #Krok_2;
      R     #H_Obr_Na_Poz_X;
      R     #H_Jedz_Na_Poz_X;
//-
      A     #Krok_1;
      AN    #Krok_2;
      =     #Trwa_Krok_1;
      S     #H_Jedz_Na_Poz_X;
      JC    j_4;
//***************************************************
//Przejdz pominiete kroki
      A     #Krok_2;
      S     #Krok_3;
//-
      A     #Krok_3;
      S     #Krok_4;
//***************************************************
//Krok 4 -Wykonaj wiazanie
      A     #H_Wiazanie_Zak_Pom;
      S     #Krok_5;
      R     #H_Wykonaj_Wiazanie;
      R     #H_Wiazanie_Zak_Pom;
      R     #H_Bindownic_Skon_Wiaz;
//-
      A     #Krok_4;
      AN    #Krok_5;
      =     #Trwa_Krok_4;
      S     #H_Wykonaj_Wiazanie;
      JC    bind;
//*****************************************************
//Krok 5 - Przerwa po zwiazaniu
      A     #H_Koniec_Pauzy;
      S     #Krok_6;
      R     #H_Poczatek_Pauzy;
      R     #H_Koniec_Pauzy;
//-
      L     T#2S;
      T     #H_Czas_Pauzy;
//-
      A     #Krok_5;
      AN    #Krok_6;
      =     #Trwa_Krok_5;
      S     #H_Poczatek_Pauzy;
      JC    wait;
//*****************************************************
//Krok 6
      A     #Krok_6;
      S     #Krok_7;
//***************************************************
//Krok 7 - Zadanie ukonczone przejdz do nastepnego zadania
      A     #Krok_7;
      JC    inc;
u_5:  NOP   0;
NETWORK
TITLE =
//Zadanie nr 6 Powrot do pozycji wyjazdu
//**************Zadanie 6 ***********************
      A     #Zadanie_6;
      JCN   u_6;
//Rozpoczecie grafu
      SET;
      S     #Krok_1;
//***************************************************
//Krok 1 - jedz na pozycje 0st 
      A     #H_Obr_Na_Poz_X;
      S     #Krok_2;
      R     #H_Obr_Na_Poz_X;
      R     #H_Jedz_Na_Poz_X;
//-
      A     #Krok_1;
      AN    #Krok_2;
      =     #Trwa_Krok_1;
      S     #H_Jedz_Na_Poz_X;
      JC    j_1;
//Pozkaz ze koniec cyklu
      A     #Krok_2;
      S     #Krok_8;
      A     #Krok_8;
      S     #o_Koniec_Cyklu;
      JC    clrs;
u_6:  NOP   0;
NETWORK
TITLE =
//Zadanie wyzerowania palety na obrotnicy
//**************Zadanie 10 ***********************
      A     #Zadanie_10;
      JCN   u_10;
//***************************************************
//Rozpoczecie grafu
      SET;
      S     #Krok_1;
//***************************************************
//Krok 1 - jedz na pozycje 0st 
      A     #H_Obr_Na_Poz_X;
      S     #Krok_2;
      R     #H_Obr_Na_Poz_X;
      R     #H_Jedz_Na_Poz_X;
//-
      A     #Krok_1;
      AN    #Krok_2;
      =     #Trwa_Krok_1;
      S     #H_Jedz_Na_Poz_X;
      JC    j_1;
//***************************************************
//Krok 2 - Jezeli tryb z pozycjonowaniem to wyœrodkuj palete
      A     #H_Paleta_Na_Srodku;
      O;
      S     #Krok_3;
      R     #H_Pozycjonuj_Srodek;
      R     #H_Paleta_Na_Srodku;
//-
      A     #Krok_2;
      AN    #Krok_3;
      =     #Trwa_Krok_2;
      S     #H_Pozycjonuj_Srodek;
      JC    res;
//-
      L     0;
      T     #io_Step_Counter;
      JU    clrs;
u_10: NOP   0;
      JU    tim;
NETWORK
TITLE =
//Puste celowo
NETWORK
TITLE =
//Rozkazy do maszyny bindujacej 
// bindowanie 
bind: NOP   0;
      A     #H_Wykonaj_Wiazanie;
      AN    #o_Bind_Start_Wiazan;
      R     #H_Bindownic_Skon_Wiaz;
      =     #H_Help_Koniec_Wiazan;
      A     #H_Wykonaj_Wiazanie;
      A     #i_Fotokomorki_Pokryte;
      S     #o_Bind_Start_Wiazan;
      A     #i_Bind_Start_Kon_Wiaz;
      FP    #Zbocze_1;
      S     #H_Wiazanie_Zak_Pom;
      R     #H_Wykonaj_Wiazanie;
      R     #o_Bind_Start_Wiazan;
      R     #H_Bindownic_Skon_Wiaz;
//bindownica wraca
      A     #i_Bind_Poloz_Podst;
      FP    #Zbocze_2;
      A     #o_Bind_Start_Wiazan;
      AN    #H_Help_Koniec_Wiazan;
      S     #H_Bindownic_Skon_Wiaz;
      A     #o_Bind_Start_Wiazan;
      A     #i_Bindownica_Auto;
      A     #H_Bindownic_Skon_Wiaz;
      AN    #H_Help_Koniec_Wiazan;
      =     #Help_Bit_1;
      CALL  #Timer_Kon_Strzalu (
           IN                       := #Help_Bit_1,
           STOP                     := #Stop_Czas_Kontrolny,
           PT                       := T#3S,
           Q_0                      := #Help_Bit_2,
           ET                       := #Czas_Aktualny);
      A     #Help_Bit_2;
      S     #H_Wiazanie_Zak_Pom;
      R     #H_Wykonaj_Wiazanie;
      R     #o_Bind_Start_Wiazan;
      R     #H_Bindownic_Skon_Wiaz;
      JU    tim;
//Pozycjonowanie Prawo
pp:   NOP   0;
      A     #H_Pozycjonuj_Prawo;
      S     #o_Pozycjonuj_Prawo;
//-
      A     #i_Pozycja_Bandy_Prawo;
      A     #i_Pozycja_Bandy_Potw;
      S     #H_Paleta_Na_Prawo;
      R     #H_Pozycjonuj_Prawo;
      R     #o_Pozycjonuj_Prawo;
      JU    tim;
//Pozycjonowanie lewo
pl:   NOP   0;
      A     #H_Pozycjonuj_Lewo;
      S     #o_Pozycjonuj_Lewo;
//-
      A     #i_Pozycja_Bandy_Lewo;
      A     #i_Pozycja_Bandy_Potw;
      S     #H_Paleta_Na_Lewo;
      R     #H_Pozycjonuj_Lewo;
      R     #o_Pozycjonuj_Lewo;
      JU    tim;
//resetowanie pozycjonowania
res:  NOP   0;
      A     #H_Pozycjonuj_Srodek;
      S     #o_Pozycjonuj_Srodek;
//-
      A     #i_Pozycja_Bandy_Srodek;
      A     #i_Pozycja_Bandy_Potw;
      S     #H_Paleta_Na_Srodku;
      R     #H_Pozycjonuj_Srodek;
      R     #o_Pozycjonuj_Srodek;
      JU    tim;
//osiagniecie pozycji 270st
j_4:  NOP   0;
      A     #H_Jedz_Na_Poz_X;
      S     #o_Jedz_Na_270st;
      A     #i_Pozycja_Obr_270st;
      A     #i_Pozycja_Obr_Osiagnieta;
      S     #H_Obr_Na_Poz_X;
      R     #o_Jedz_Na_270st;
      R     #H_Jedz_Na_Poz_X;
      JU    tim;
//osiagniecie pozycji 180st
j_3:  NOP   0;
      A     #H_Jedz_Na_Poz_X;
      S     #o_Jedz_Na_180st;
      A     #i_Pozycja_Obr_180st;
      A     #i_Pozycja_Obr_Osiagnieta;
      S     #H_Obr_Na_Poz_X;
      R     #o_Jedz_Na_180st;
      R     #H_Jedz_Na_Poz_X;
      JU    tim;
//osiagniecie pozycji 90st
j_2:  NOP   0;
      A     #H_Jedz_Na_Poz_X;
      S     #o_Jedz_Na_90st;
      A     #i_Pozycja_Obr_90st;
      A     #i_Pozycja_Obr_Osiagnieta;
      S     #H_Obr_Na_Poz_X;
      R     #o_Jedz_Na_90st;
      R     #H_Jedz_Na_Poz_X;
      JU    tim;
//osiagniecie pozycji 0st
j_1:  NOP   0;
      A     #H_Jedz_Na_Poz_X;
      S     #o_Jedz_Na_0st;
      A     #i_Pozycja_Obr_0st;
      A     #i_Pozycja_Obr_Osiagnieta;
      S     #H_Obr_Na_Poz_X;
      R     #o_Jedz_Na_0st;
      R     #H_Jedz_Na_Poz_X;
      JU    tim;
//zerowanie licznika
zer:  NOP   0;
      L     0;
      T     #io_Step_Counter;
      JU    clrs;
//Zwiekszenie licznika krokow o 1  
inc:  NOP   0;
      L     #io_Step_Counter;
      L     1;
      +I;
      T     #io_Step_Counter;
clrs: SET;
//resetowanie bitow pracy programu
//k1
      R     #H_Jedz_Na_Poz_X;
      R     #H_Obr_Na_Poz_X;
//k2
      R     #H_Pozycjonuj_Srodek;
      R     #H_Paleta_Na_Srodku;
//k3
      R     #H_Pozycjonuj_Prawo;
      R     #H_Paleta_Na_Prawo;
//k4
      R     #H_Pozycjonuj_Lewo;
      R     #H_Paleta_Na_Lewo;
//k5
      R     #H_Wykonaj_Wiazanie;
      R     #H_Wiazanie_Zak_Pom;
      R     #H_Wykonaj_Wiazanie;
      R     #H_Bindownic_Skon_Wiaz;
      R     #H_Wiazanie_Zak_Pom;
//k6
      R     #H_Poczatek_Pauzy;
      R     #H_Koniec_Pauzy;
      R     #H_Bit_Pauzy;
//Bt
      R     #H_Bindownic_Skon_Wiaz;
//-
      R     #Krok_1;
      R     #Krok_2;
      R     #Krok_3;
      R     #Krok_4;
      R     #Krok_5;
      R     #Krok_6;
      R     #Krok_7;
      R     #Krok_8;
      R     #Krok_9;
//-
      R     #Trwa_Krok_1;
      R     #Trwa_Krok_2;
      R     #Trwa_Krok_3;
      R     #Trwa_Krok_4;
      R     #Trwa_Krok_5;
      R     #Trwa_Krok_6;
      R     #Trwa_Krok_7;
      R     #Trwa_Krok_8;
      R     #Trwa_Krok_9;
//-
      R     #o_Pozycjonuj_Lewo;
      R     #o_Pozycjonuj_Prawo;
      R     #o_Pozycjonuj_Srodek;
      R     #o_Jedz_Na_0st;
      R     #o_Jedz_Na_90st;
      R     #o_Jedz_Na_180st;
      R     #o_Jedz_Na_270st;
      R     #o_Bind_Start_Wiazan;
      JU    tim;
//Czas Pauzy
wait: NOP   0;
      CALL  #Timer_Pauzy (
           IN                       := #H_Bit_Pauzy,
           STOP                     := #Stop_Czas_Kontrolny,
           PT                       := #H_Czas_Pauzy,
           Q_0                      := #Help_Bit_1,
           ET                       := #Czas_Aktualny);
      A     #H_Poczatek_Pauzy;
      S     #H_Bit_Pauzy;
      A     #Help_Bit_1;
      R     #H_Poczatek_Pauzy;
      R     #H_Bit_Pauzy;
      S     #H_Koniec_Pauzy;
      JU    tim;
NETWORK
TITLE =
//Czas kontrolny poszczegolnych krokow
//**************************************************
//Kontynuacja programu sprawdzenie czasow tranzycji
tim:  NOP   0;
NETWORK
TITLE =
//Sprawdzenie czy czas nie przeszedl za daleko
      SET;
      R     #H_Blad;
NETWORK
TITLE =
//Zezwolenie na prace bindownicy
//0st ok
      AN    #H_Blad;
      A     #i_Pozycja_Obr_0st;
      AN    #i_Pozycja_Bandy_Lewo;
      A     #i_Fotokomorki_Pokryte;
      =     #H_Pozycja_0_st_ok;
//90st ok
      A     #i_Pozycja_Obr_90st;
      AN    #H_Blad;
      A     #i_Fotokomorki_Pokryte;
      =     #H_Pozycja_90_st_ok;
//180st
      AN    #H_Blad;
      A     #i_Pozycja_Obr_180st;
      AN    #i_Pozycja_Bandy_Prawo;
      A     #i_Fotokomorki_Pokryte;
      =     #H_Pozycja_180_st_ok;
//270st
      AN    #H_Blad;
      A     #i_Pozycja_Obr_270st;
      A     #i_Fotokomorki_Pokryte;
      =     #H_Pozycja_270_st_ok;
//Zezwolenie na prace bindownicy
      O     #H_Pozycja_0_st_ok;
      O     #H_Pozycja_90_st_ok;
      O     #H_Pozycja_180_st_ok;
      O     #H_Pozycja_270_st_ok;
      A     #i_Marka_Bezpieczenstwa;
      =     #o_Bind_Zez_Na_Prace;
END_FUNCTION_BLOCK

FUNCTION_BLOCK "Wybranie_Wjazdu"	// FB 50
VERSION : 0.1
VAR_INPUT
  Zajetosc_1_Lini : BOOL ;
  Zajetosc_2_Lini : BOOL ;
  Zezwolenie_Do_1_Lini : BOOL ;
  Zezwolenie_Do_2_Lini : BOOL ;
  Zabierz_Od_1_Lini : BOOL ;
  Zabierz_Od_2_Lini : BOOL ;
  Silniki_Nie_Pracuja : BOOL ;
END_VAR
VAR_IN_OUT
  Blokada_Kierunku_1 : BOOL ;
  Blokada_Kierunku_2 : BOOL ;
  Blokada : BOOL ;
END_VAR
VAR
  Czas_Kontrolny : SFB 4;
END_VAR
VAR_TEMP
  Temp_Help_1 : BOOL ;
  Temp_Help_2 : BOOL ;
END_VAR
BEGIN
NETWORK
TITLE =
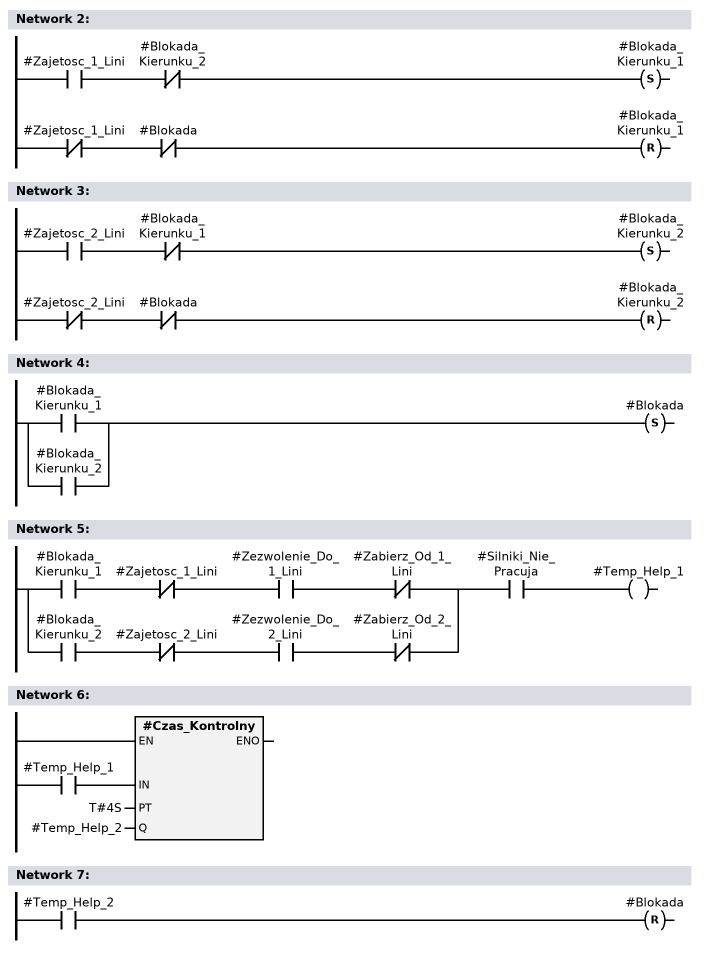
NETWORK
TITLE =
//Zarezerwowanie poboru palety z pierwszej lini
      A     #Zajetosc_1_Lini;
      AN    #Blokada_Kierunku_2;
      S     #Blokada_Kierunku_1;
      AN    #Zajetosc_1_Lini;
      AN    #Blokada;
      R     #Blokada_Kierunku_1;
      NOP   0;
NETWORK
TITLE =
//Zarezewowanie poboru palety z durgiej lini
      A     #Zajetosc_2_Lini;
      AN    #Blokada_Kierunku_1;
      S     #Blokada_Kierunku_2;
      AN    #Zajetosc_2_Lini;
      AN    #Blokada;
      R     #Blokada_Kierunku_2;
      NOP   0;
NETWORK
TITLE =
      A(;
      O     #Blokada_Kierunku_1;
      O     #Blokada_Kierunku_2;
      );
      S     #Blokada;
      NOP   0;
      NOP   0;
NETWORK
TITLE =
      A(;
      A     #Blokada_Kierunku_1;
      AN    #Zajetosc_1_Lini;
      A     #Zezwolenie_Do_1_Lini;
      AN    #Zabierz_Od_1_Lini;
      O;
      A     #Blokada_Kierunku_2;
      AN    #Zajetosc_2_Lini;
      A     #Zezwolenie_Do_2_Lini;
      AN    #Zabierz_Od_2_Lini;
      );
      A     #Silniki_Nie_Pracuja;
      =     #Temp_Help_1;
NETWORK
TITLE =
//Czas kontolny po ktorym nastepuje ponowne wybranie kierunku wjazdu
      A     #Temp_Help_1;
      =     L 1.0;
      BLD   103;
      CALL  #Czas_Kontrolny (
           IN                       := L 1.0,
           PT                       := T#4S,
           Q                        := #Temp_Help_2);
      NOP   0;
NETWORK
TITLE =
      A     #Temp_Help_2;
      R     #Blokada;
END_FUNCTION_BLOCK

FUNCTION_BLOCK "Obr_Na_Poz_1"	// FB 51
VERSION : 0.1
VAR_INPUT
  Jedz_Na_90st : BOOL ;
  Jedz_Na_0st : BOOL ;
  Czujnik_90st : BOOL ;
  Czujnik_0st : BOOL ;
  Czujnik_Ham_90st : BOOL ;
  Czujnik_Ham_0st : BOOL ;
  Odblowuj_Obrotnice : BOOL ;
END_VAR
VAR_OUTPUT
  Na_Pozycji_0st : BOOL ;	//Obrotnica na pozycji 0 stopni
  Na_Pozycji_90st : BOOL ;	//Obrotnica na pozycji 90 stopni
  Motor_Wolno : BOOL ;
  Odblokowanie_Rolek : BOOL ;
END_VAR
VAR_IN_OUT
  Talerz_w_Lewo : BOOL ;
  Talerz_w_Prawo : BOOL ;
END_VAR
VAR
  Czas_Dojscia : SFB 4;
  Czas_Startu : SFB 4;
  Help_Start : BOOL ;
END_VAR
VAR_TEMP
  Help_1 : BOOL ;
END_VAR
BEGIN
NETWORK
TITLE =
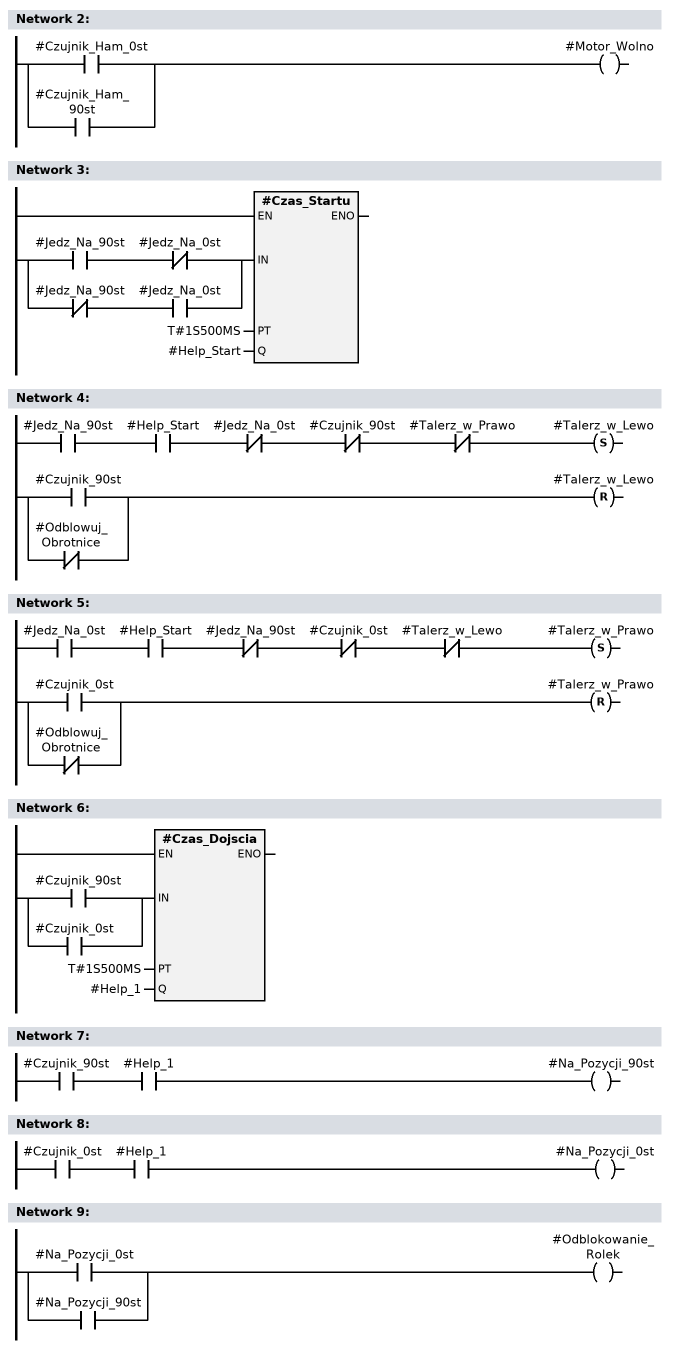
NETWORK
TITLE =
//Motor wolno gdy czujniki hamowania
      O     #Czujnik_Ham_0st;
      O     #Czujnik_Ham_90st;
      =     #Motor_Wolno;
NETWORK
TITLE =
      A(;
      A     #Jedz_Na_90st;
      AN    #Jedz_Na_0st;
      O;
      AN    #Jedz_Na_90st;
      A     #Jedz_Na_0st;
      );
      =     L 1.0;
      BLD   103;
      CALL  #Czas_Startu (
           IN                       := L 1.0,
           PT                       := T#1S500MS,
           Q                        := #Help_Start);
      NOP   0;
NETWORK
TITLE =
      A     #Jedz_Na_90st;
      A     #Help_Start;
      AN    #Jedz_Na_0st;
      AN    #Czujnik_90st;
      AN    #Talerz_w_Prawo;
      S     #Talerz_w_Lewo;
      A(;
      O     #Czujnik_90st;
      ON    #Odblowuj_Obrotnice;
      );
      R     #Talerz_w_Lewo;
      NOP   0;
NETWORK
TITLE =
      A     #Jedz_Na_0st;
      A     #Help_Start;
      AN    #Jedz_Na_90st;
      AN    #Czujnik_0st;
      AN    #Talerz_w_Lewo;
      S     #Talerz_w_Prawo;
      A(;
      O     #Czujnik_0st;
      ON    #Odblowuj_Obrotnice;
      );
      R     #Talerz_w_Prawo;
      NOP   0;
NETWORK
TITLE =
      A(;
      O     #Czujnik_90st;
      O     #Czujnik_0st;
      );
      =     L 1.0;
      BLD   103;
      CALL  #Czas_Dojscia (
           IN                       := L 1.0,
           PT                       := T#1S500MS,
           Q                        := #Help_1);
      NOP   0;
NETWORK
TITLE =
      A     #Czujnik_90st;
      A     #Help_1;
      =     #Na_Pozycji_90st;
NETWORK
TITLE =
      A     #Czujnik_0st;
      A     #Help_1;
      =     #Na_Pozycji_0st;
NETWORK
TITLE =
//Odblokowanie napedu rolkowego
      O     #Na_Pozycji_0st;
      O     #Na_Pozycji_90st;
      =     #Odblokowanie_Rolek;
END_FUNCTION_BLOCK

FUNCTION_BLOCK "Obr_Na_Poz_2"	// FB 52
//Funkcja sterujaca banda obrotowa. Programowana na jazde do roznych celow
VERSION : 0.1
VAR_INPUT
  Jedz_Na_90st : BOOL ;
  Jedz_Na_0st : BOOL ;
  Jedz_Na_45_st : BOOL ;
  Czujnik_90st : BOOL ;
  Czujnik_0st : BOOL ;
  Czujnik_45st_1 : BOOL ;
  Czujnik_45st_2 : BOOL ;
  Czujnik_Ham_90st : BOOL ;
  Czujnik_Ham_0st : BOOL ;
  Odblowuj_Obrotnice : BOOL ;
  Silownik_Bezpiecczny : BOOL ;
END_VAR
VAR_OUTPUT
  Na_Pozycji_0st : BOOL ;	//Obrotnica na pozycji 0 stopni
  Na_Pozycji_90st : BOOL ;	//Obrotnica na pozycji 90 stopni
  Na_Pozycji_45_st : BOOL ;
  Motor_Wolno : BOOL ;
  Odblokowanie_Rolek : BOOL ;
END_VAR
VAR_IN_OUT
  Talerz_w_Lewo : BOOL ;
  Talerz_w_Prawo : BOOL ;
END_VAR
VAR
  Czas_Dojscia : SFB 4;
  Czas_Startu : SFB 4;
  Help_Start : BOOL ;
END_VAR
VAR_TEMP
  Help_1 : BOOL ;
END_VAR
BEGIN
NETWORK
TITLE =
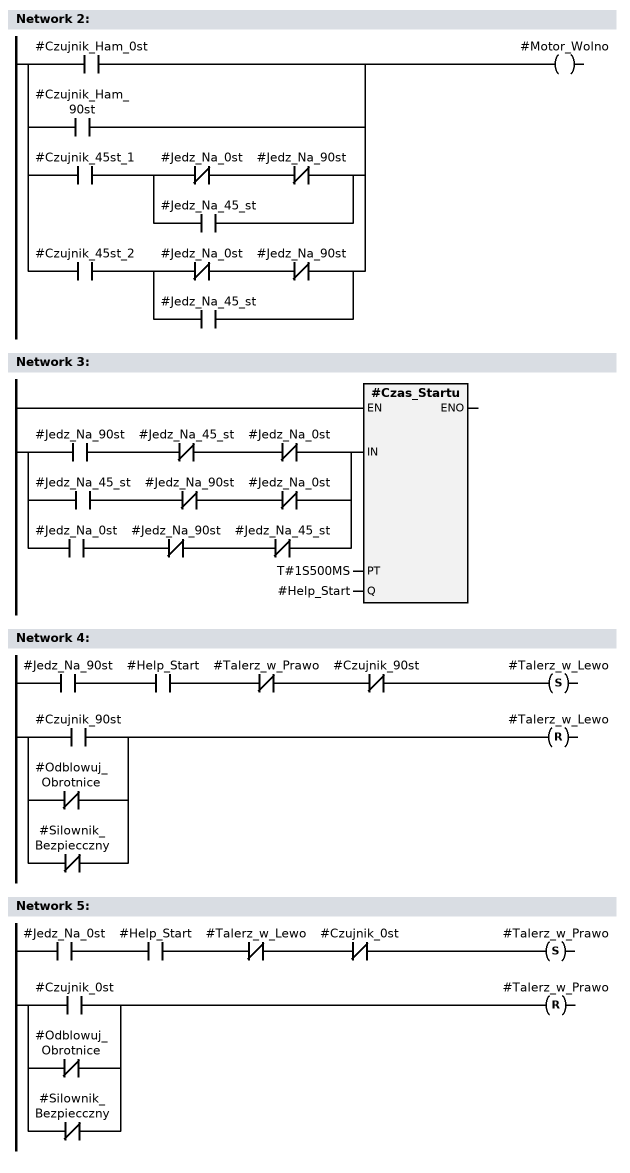
NETWORK
TITLE =
//Motor wolno gdy czujniki hamowania
      O     #Czujnik_Ham_0st;
      O     #Czujnik_Ham_90st;
      O;
      A     #Czujnik_45st_1;
      A(;
      AN    #Jedz_Na_0st;
      AN    #Jedz_Na_90st;
      O     #Jedz_Na_45_st;
      );
      O;
      A     #Czujnik_45st_2;
      A(;
      AN    #Jedz_Na_0st;
      AN    #Jedz_Na_90st;
      O     #Jedz_Na_45_st;
      );
      =     #Motor_Wolno;
NETWORK
TITLE =
      A(;
      A     #Jedz_Na_90st;
      AN    #Jedz_Na_45_st;
      AN    #Jedz_Na_0st;
      O;
      A     #Jedz_Na_45_st;
      AN    #Jedz_Na_90st;
      AN    #Jedz_Na_0st;
      O;
      A     #Jedz_Na_0st;
      AN    #Jedz_Na_90st;
      AN    #Jedz_Na_45_st;
      );
      =     L 1.0;
      BLD   103;
      CALL  #Czas_Startu (
           IN                       := L 1.0,
           PT                       := T#1S500MS,
           Q                        := #Help_Start);
      NOP   0;
NETWORK
TITLE =
      A     #Jedz_Na_90st;
      A     #Help_Start;
      AN    #Talerz_w_Prawo;
      AN    #Czujnik_90st;
      S     #Talerz_w_Lewo;
      A(;
      O     #Czujnik_90st;
      ON    #Odblowuj_Obrotnice;
      ON    #Silownik_Bezpiecczny;
      );
      R     #Talerz_w_Lewo;
      NOP   0;
NETWORK
TITLE =
      A     #Jedz_Na_0st;
      A     #Help_Start;
      AN    #Talerz_w_Lewo;
      AN    #Czujnik_0st;
      S     #Talerz_w_Prawo;
      A(;
      O     #Czujnik_0st;
      ON    #Odblowuj_Obrotnice;
      ON    #Silownik_Bezpiecczny;
      );
      R     #Talerz_w_Prawo;
      NOP   0;
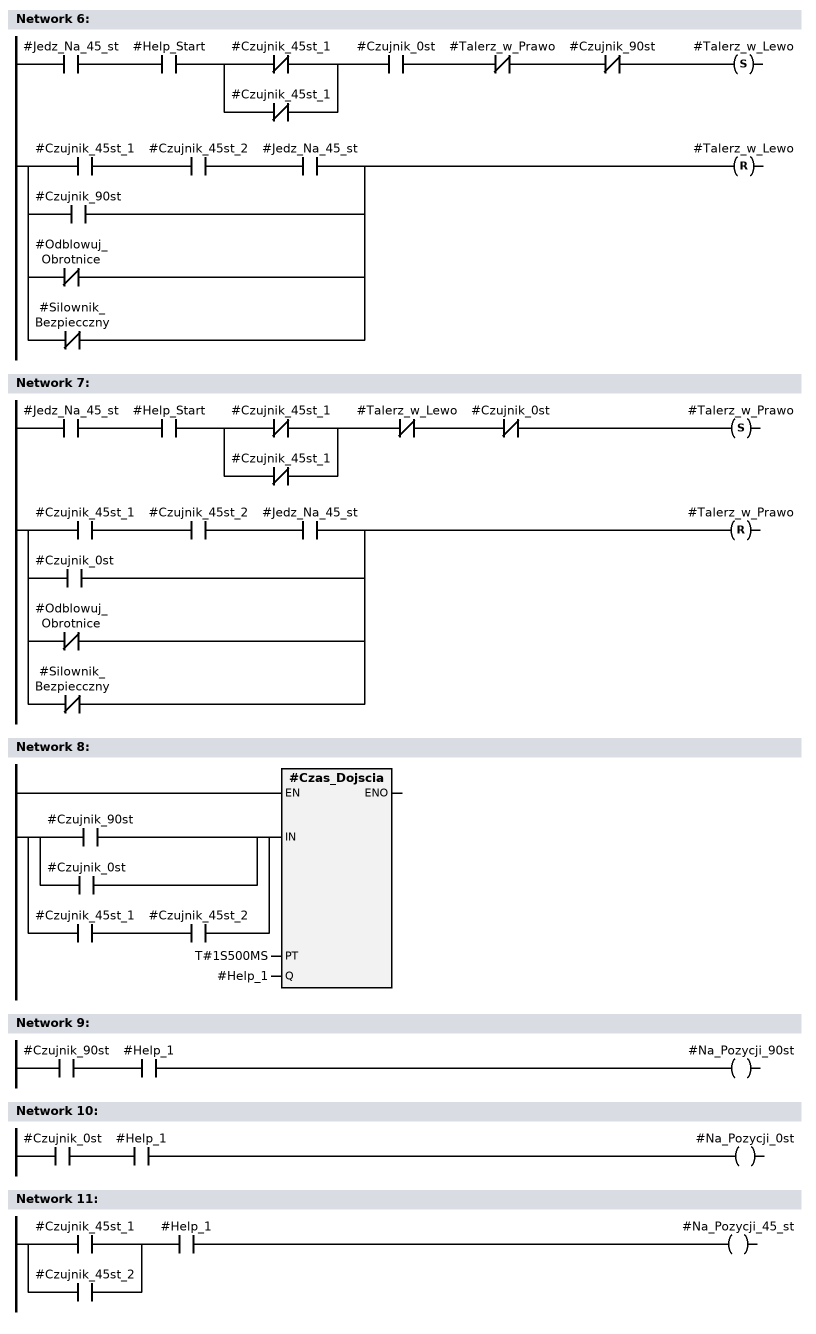
NETWORK
TITLE =
//Jazda na punkt 45st
      A     #Jedz_Na_45_st;
      A     #Help_Start;
      A(;
      ON    #Czujnik_45st_1;
      ON    #Czujnik_45st_1;
      );
      A     #Czujnik_0st;
      AN    #Talerz_w_Prawo;
      AN    #Czujnik_90st;
      S     #Talerz_w_Lewo;
      A(;
      A     #Czujnik_45st_1;
      A     #Czujnik_45st_2;
      A     #Jedz_Na_45_st;
      O     #Czujnik_90st;
      ON    #Odblowuj_Obrotnice;
      ON    #Silownik_Bezpiecczny;
      );
      R     #Talerz_w_Lewo;
      NOP   0;
NETWORK
TITLE =
//celowo brak czujnika 90st w ladzie
      A     #Jedz_Na_45_st;
      A     #Help_Start;
      A(;
      ON    #Czujnik_45st_1;
      ON    #Czujnik_45st_1;
      );
      AN    #Talerz_w_Lewo;
      AN    #Czujnik_0st;
      S     #Talerz_w_Prawo;
      A(;
      A     #Czujnik_45st_1;
      A     #Czujnik_45st_2;
      A     #Jedz_Na_45_st;
      O     #Czujnik_0st;
      ON    #Odblowuj_Obrotnice;
      ON    #Silownik_Bezpiecczny;
      );
      R     #Talerz_w_Prawo;
      NOP   0;
NETWORK
TITLE =
//Opoznienie przyjcia informacji o dojezdzie na pozycje
      A(;
      O     #Czujnik_90st;
      O     #Czujnik_0st;
      O;
      A     #Czujnik_45st_1;
      A     #Czujnik_45st_2;
      );
      =     L 1.0;
      BLD   103;
      CALL  #Czas_Dojscia (
           IN                       := L 1.0,
           PT                       := T#1S500MS,
           Q                        := #Help_1);
      NOP   0;
NETWORK
TITLE =
      A     #Czujnik_90st;
      A     #Help_1;
      =     #Na_Pozycji_90st;
NETWORK
TITLE =
      A     #Czujnik_0st;
      A     #Help_1;
      =     #Na_Pozycji_0st;
NETWORK
TITLE =
      A(;
      O     #Czujnik_45st_1;
      O     #Czujnik_45st_2;
      );
      A     #Help_1;
      =     #Na_Pozycji_45_st;
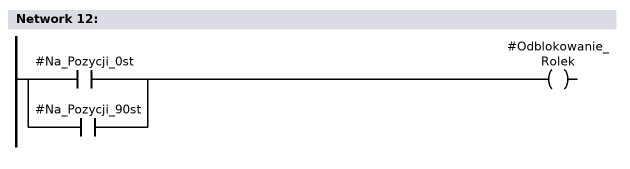
NETWORK
TITLE =
//Odblokowanie napedu rolkowego
      O     #Na_Pozycji_0st;
      O     #Na_Pozycji_90st;
      =     #Odblokowanie_Rolek;
END_FUNCTION_BLOCK

FUNCTION_BLOCK "Obr_Na_Poz_4"	// FB 54
//Funkcja sterujaca banda obrotowa. Programowana na jazde do roznych celow. 
//Zachowuje ona mo¿liwoœæ jazdy na 4 pozycje w zale¿noœci od po³o¿enia 
//inicjatorów 
//Kieunek jest wybierany ze wzgledu na wartosc liczbowa przyporzadkowana do 
//czujnikow. 
//
//0st_1- 1 czunik ostateczny oraz czujnik pozycji 0 stopni
//0st_2- 2 czujnik hamowania
//90st_1- 89 czujnik hamowania
//90st_2- 90 czujnik pozycji 90 stopni
//180st_1-179 czujnik hamowania 
//180st_2-180 czujnil pozycji 180 stopni
//270st_1-269 czujnik hamowania 
//270st_2-270 czujnik ostateczny oraz czujnik pozycji 270 stopni
//
//Czujniki ustawiane sa tak by przy obrocie we wlasciwym kierunku pracy najpierw 
//atakowany by³ czujnik hamowania a nastepnie czujnik pozycji docelowej
//Wyjatiem jest czujnik 0st(bo element startowy).
//
VERSION : 0.1
VAR_INPUT
  i_Marka_Bezpieczenstwa : BOOL ;
  i_Auto_Reczny : BOOL ;	//Auto-1,Reczny-0
  Zawsze_True : BOOL ;
  Jedz_Na_0st : BOOL ;
  Jedz_Na_90st : BOOL ;
  Jedz_Na_180st : BOOL ;
  Jedz_Na_270_st : BOOL ;
  Czujnik_0st_1 : BOOL ;
  Czujnik_0st_2 : BOOL ;
  Czujnik_90st_1 : BOOL ;
  Czujnik_90st_2 : BOOL ;
  Czujnik_180st_1 : BOOL ;
  Czujnik_180st_2 : BOOL ;
  Czujnik_270st_1 : BOOL ;
  Czujnik_270st_2 : BOOL ;
  Przycisk_Lewo : BOOL ;
  Przycisk_Prawo : BOOL ;
  s_Zez_Na_Obr : BOOL ;
  s_Ramie_Bind_w_Tyle : BOOL ;
END_VAR
VAR_OUTPUT
  Na_Pozycji_0st : BOOL ;	//Obrotnica na pozycji 0 stopni
  Na_Pozycji_90st : BOOL ;	//Obrotnica na pozycji 90 stopni
  Na_Pozycji_180st : BOOL ;
  Na_Pozycji_270st : BOOL ;
  Poz_Osiagnieta : BOOL ;	//Pozycja zadana osiagnieta
  s_Zez_Na_Rolki : BOOL ;	//Rolki odblowkowne je¿eli bindownica w poziomie do lini
  Motor_Wolno : BOOL ;
END_VAR
VAR_IN_OUT
  Talerz_w_Lewo : BOOL ;
  Talerz_w_Prawo : BOOL ;
  Pozycja : INT ;
END_VAR
VAR
  Czas_Dojscia : SFB 4;
  Czas_Startu : SFB 4;
  Help_Start : BOOL ;
  Help_Poz_0st : BOOL ;
  Help_Poz_90st : BOOL ;
  Help_Poz_180st : BOOL ;
  Help_Poz_270st : BOOL ;
  Help_A_Talerz_w_Prawo : BOOL ;	//CW
  Help_A_Talerz_w_Lewo : BOOL ;	//CCW
  Help_A_Motor_Wolno : BOOL ;
  Help_H_Talerz_w_Prawo : BOOL ;	//CW
  Help_H_Talerz_w_Lewo : BOOL ;	//CCW
  Help_H_Motor_Wolno : BOOL ;
  Help_Zbocze_0 : BOOL ;
  Help_Zbocze_1 : BOOL ;
  Help_Zbocze_2 : BOOL ;
  Help_Zbocze_3 : BOOL ;
  Help_Zbocze_4 : BOOL ;
  Silniki_nie_pracuja : BOOL ;
  Help_Opoznienie : BOOL ;
  Stop_Czas : BOOL ;
  help_18 : BOOL ;
  help_19 : BOOL ;
  help_20 : BOOL ;
END_VAR
VAR_TEMP
  Help_1 : BOOL ;
END_VAR
BEGIN
NETWORK
TITLE =
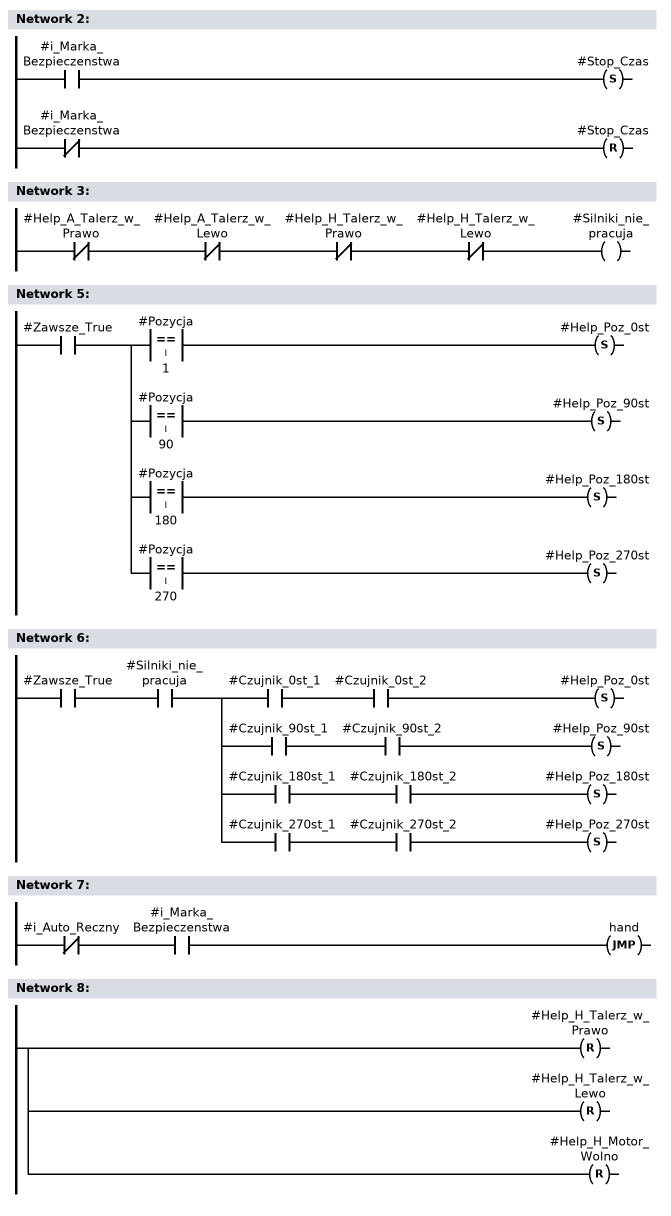
NETWORK
TITLE =
//ten network celowo jest wolny 
      A     #i_Marka_Bezpieczenstwa;
      S     #Stop_Czas;
      AN    #i_Marka_Bezpieczenstwa;
      R     #Stop_Czas;
NETWORK
TITLE =
//Sprawdzenie czy silniki nie pracuja 
      AN    #Help_A_Talerz_w_Prawo;
      AN    #Help_A_Talerz_w_Lewo;
      AN    #Help_H_Talerz_w_Prawo;
      AN    #Help_H_Talerz_w_Lewo;
      =     #Silniki_nie_pracuja;
NETWORK
TITLE =
      L     #Pozycja;
//********pozycja 0 stopni
//Pozycj 0 stopni obrotnica w pozycji wjazdu
      A     #Czujnik_0st_1;
      JCN   et_1;
      L     1;
      JU    poz;
et_1: NOP   0;
//zalaczony czujnik hamowania  samodzielnie
      A     #Czujnik_0st_2;
      AN    #Czujnik_0st_1;
      JCN   et_2;
      L     2;
      JU    poz;
et_2: NOP   0;
//********pozycja 90 stopni
//w kierunku cw najazd normalny z hamowaniem 
//w kierunku ccw najzd z minieciem pozycji + powrot
//czujnik 90 stopni hamowanie / w prawo
      O     #Help_A_Talerz_w_Prawo;
      O     #Help_H_Talerz_w_Prawo;
      A     #Czujnik_90st_1;
      AN    #Czujnik_90st_2;
      JCN   et_3;
      L     89;
      JU    poz;
et_3: NOP   0;
//czujnik 90 stopni pozycja  / w prawo
      O     #Help_A_Talerz_w_Prawo;
      O     #Help_H_Talerz_w_Prawo;
      A     #Czujnik_90st_2;
      JCN   et_4;
      L     90;
      JU    poz;
et_4: NOP   0;
//czujnik 90 stopni / w lewo
      O     #Help_A_Talerz_w_Lewo;
      O     #Help_H_Talerz_w_Lewo;
      A     #Czujnik_90st_2;
      JCN   e_13;
      L     91;
      JU    poz;
e_13: NOP   0;
//czujnik hamowania 90 stopni w lewo 
      O     #Help_A_Talerz_w_Lewo;
      O     #Help_H_Talerz_w_Lewo;
      A     #Czujnik_90st_1;
      AN    #Czujnik_90st_2;
      JCN   e_14;
      L     88;
      JU    poz;
e_14: NOP   0;
//********pozycja 180 stopni
//w kierunku ccw najzd z minieciem pozycji + powrot
//czujnik 180 stopni hamowanie
      O     #Help_A_Talerz_w_Prawo;
      O     #Help_H_Talerz_w_Prawo;
      A     #Czujnik_180st_1;
      AN    #Czujnik_180st_2;
      JCN   et_6;
      L     179;
      JU    poz;
et_6: NOP   0;
//czujnik 180 stopni pozycja
      O     #Help_A_Talerz_w_Prawo;
      O     #Help_H_Talerz_w_Prawo;
      A     #Czujnik_180st_2;
      JCN   et_7;
      L     180;
      JU    poz;
et_7: NOP   0;
//czujnik 180 stopni / w lewo
      O     #Help_A_Talerz_w_Lewo;
      O     #Help_H_Talerz_w_Lewo;
      A     #Czujnik_180st_2;
      JCN   e_16;
      L     181;
      JU    poz;
e_16: NOP   0;
//czujnik hamowania 180stopni w lewo 
      O     #Help_A_Talerz_w_Lewo;
      O     #Help_H_Talerz_w_Lewo;
      A     #Czujnik_180st_1;
      AN    #Czujnik_180st_2;
      JCN   e_17;
      L     178;
      JU    poz;
e_17: NOP   0;
//********pozycja 270 stopni
//270 stopni pozycja hamowania
      A     #Czujnik_270st_1;
      AN    #Czujnik_270st_2;
      JCN   et_8;
      L     269;
      JU    poz;
et_8: NOP   0;
//czujnik 270 stopni pozycja
      A     #Czujnik_270st_2;
      JCN   et_9;
      L     270;
      JU    poz;
et_9: NOP   0;
//Przypisanie wartosci pozycji
poz:  NOP   0;
      T     #Pozycja;
//sprawdz czy wartosci mieszcza sie w zakresie
      O(;
      L     #Pozycja;
      L     1;
      <I;
      );
      O(;
      L     #Pozycja;
      L     270;
      >I;
      );
      JCN   cv;
      L     100;
      T     #Pozycja;
cv:   NOP   0;
NETWORK
TITLE =
//Sprawdzenie pozycji dla recznego
      A     #Zawsze_True;
      =     L 1.0;
      A     L 1.0;
      A(;
      L     #Pozycja;
      L     1;
      ==I;
      );
      S     #Help_Poz_0st;
      A     L 1.0;
      A(;
      L     #Pozycja;
      L     90;
      ==I;
      );
      S     #Help_Poz_90st;
      A     L 1.0;
      A(;
      L     #Pozycja;
      L     180;
      ==I;
      );
      S     #Help_Poz_180st;
      A     L 1.0;
      A(;
      L     #Pozycja;
      L     270;
      ==I;
      );
      S     #Help_Poz_270st;
NETWORK
TITLE =
////Warunkowe przypisanie pozycji po glebszym bledzie
      A     #Zawsze_True;
      A     #Silniki_nie_pracuja;
      =     L 1.0;
      A     L 1.0;
      A     #Czujnik_0st_1;
      A     #Czujnik_0st_2;
      S     #Help_Poz_0st;
      A     L 1.0;
      A     #Czujnik_90st_1;
      A     #Czujnik_90st_2;
      S     #Help_Poz_90st;
      A     L 1.0;
      A     #Czujnik_180st_1;
      A     #Czujnik_180st_2;
      S     #Help_Poz_180st;
      A     L 1.0;
      A     #Czujnik_270st_1;
      A     #Czujnik_270st_2;
      S     #Help_Poz_270st;
NETWORK
TITLE =
//jazda na pozycje zadana
//skocz jezeli tryb reczny
      AN    #i_Auto_Reczny;
      A     #i_Marka_Bezpieczenstwa;
      JC    hand;
NETWORK
TITLE =
//Kasowanie bitow z trybu recznego 
      SET;
      R     #Help_H_Talerz_w_Prawo;
      R     #Help_H_Talerz_w_Lewo;
      R     #Help_H_Motor_Wolno;
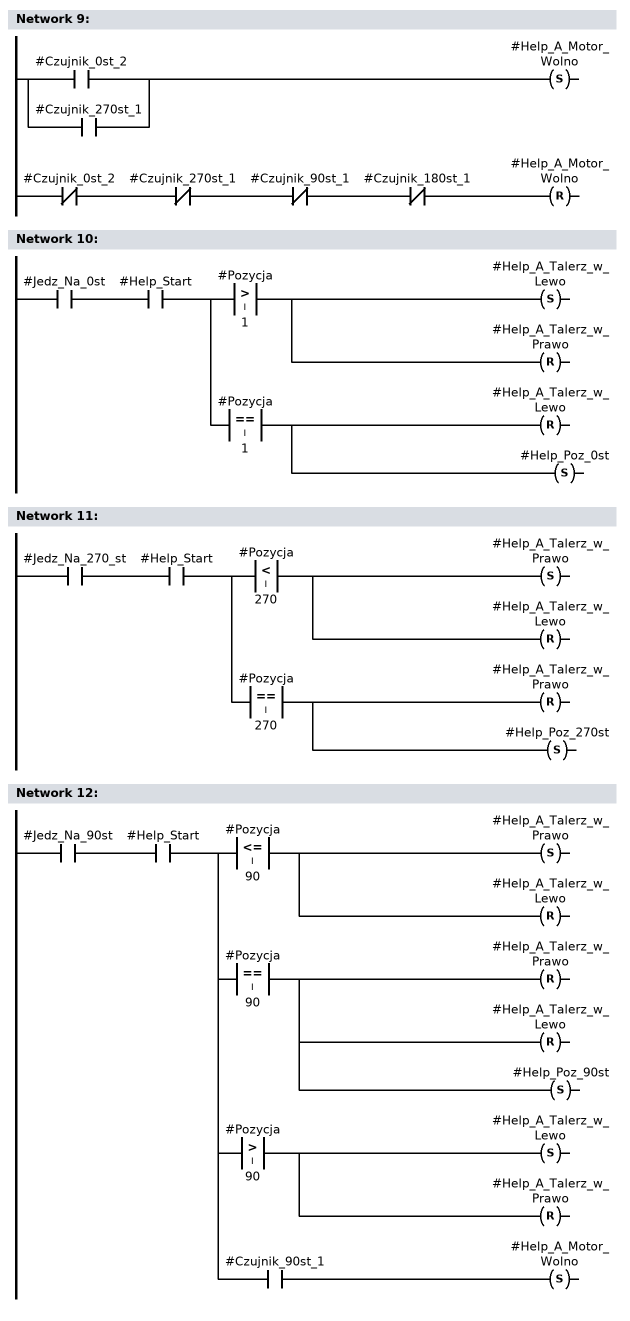
NETWORK
TITLE =
//Zalaczenie trybu wolnego. Wylaczony gdy zaden z czujnikow nie jest zalaczony
      A(;
      O     #Czujnik_0st_2;
      O     #Czujnik_270st_1;
      );
      S     #Help_A_Motor_Wolno;
      AN    #Czujnik_0st_2;
      AN    #Czujnik_270st_1;
      AN    #Czujnik_90st_1;
      AN    #Czujnik_180st_1;
      R     #Help_A_Motor_Wolno;
      NOP   0;
NETWORK
TITLE =
//Jazda na pozycje 0 st
//
      A     #Jedz_Na_0st;
      A     #Help_Start;
      =     L 1.0;
      A     L 1.0;
      A(;
      L     #Pozycja;
      L     1;
      >I;
      );
      S     #Help_A_Talerz_w_Lewo;
      R     #Help_A_Talerz_w_Prawo;
      A     L 1.0;
      A(;
      L     #Pozycja;
      L     1;
      ==I;
      );
      R     #Help_A_Talerz_w_Lewo;
      S     #Help_Poz_0st;
NETWORK
TITLE =
//Jazda na pozycje 270st 
//
      A     #Jedz_Na_270_st;
      A     #Help_Start;
      =     L 1.0;
      A     L 1.0;
      A(;
      L     #Pozycja;
      L     270;
      <I;
      );
      S     #Help_A_Talerz_w_Prawo;
      R     #Help_A_Talerz_w_Lewo;
      A     L 1.0;
      A(;
      L     #Pozycja;
      L     270;
      ==I;
      );
      R     #Help_A_Talerz_w_Prawo;
      S     #Help_Poz_270st;
NETWORK
TITLE =
//Jazda na 90 st od strony lewej i od strony prawej. Gdy najazd od strony lewej 
//najpierw jest hamowanie talerza nastepnie zatrzymanie. Gdy najazd od strony 
//prawej nastepuje miniecie czujnika nastepnie zatrzymanie i cofniecie
//
//
      A     #Jedz_Na_90st;
      A     #Help_Start;
      =     L 1.0;
      A     L 1.0;
      A(;
      L     #Pozycja;
      L     90;
      <=I;
      );
      S     #Help_A_Talerz_w_Prawo;
      R     #Help_A_Talerz_w_Lewo;
      A     L 1.0;
      A(;
      L     #Pozycja;
      L     90;
      ==I;
      );
      R     #Help_A_Talerz_w_Prawo;
      R     #Help_A_Talerz_w_Lewo;
      S     #Help_Poz_90st;
      A     L 1.0;
      A(;
      L     #Pozycja;
      L     90;
      >I;
      );
      S     #Help_A_Talerz_w_Lewo;
      R     #Help_A_Talerz_w_Prawo;
      A     L 1.0;
      A     #Czujnik_90st_1;
      S     #Help_A_Motor_Wolno;
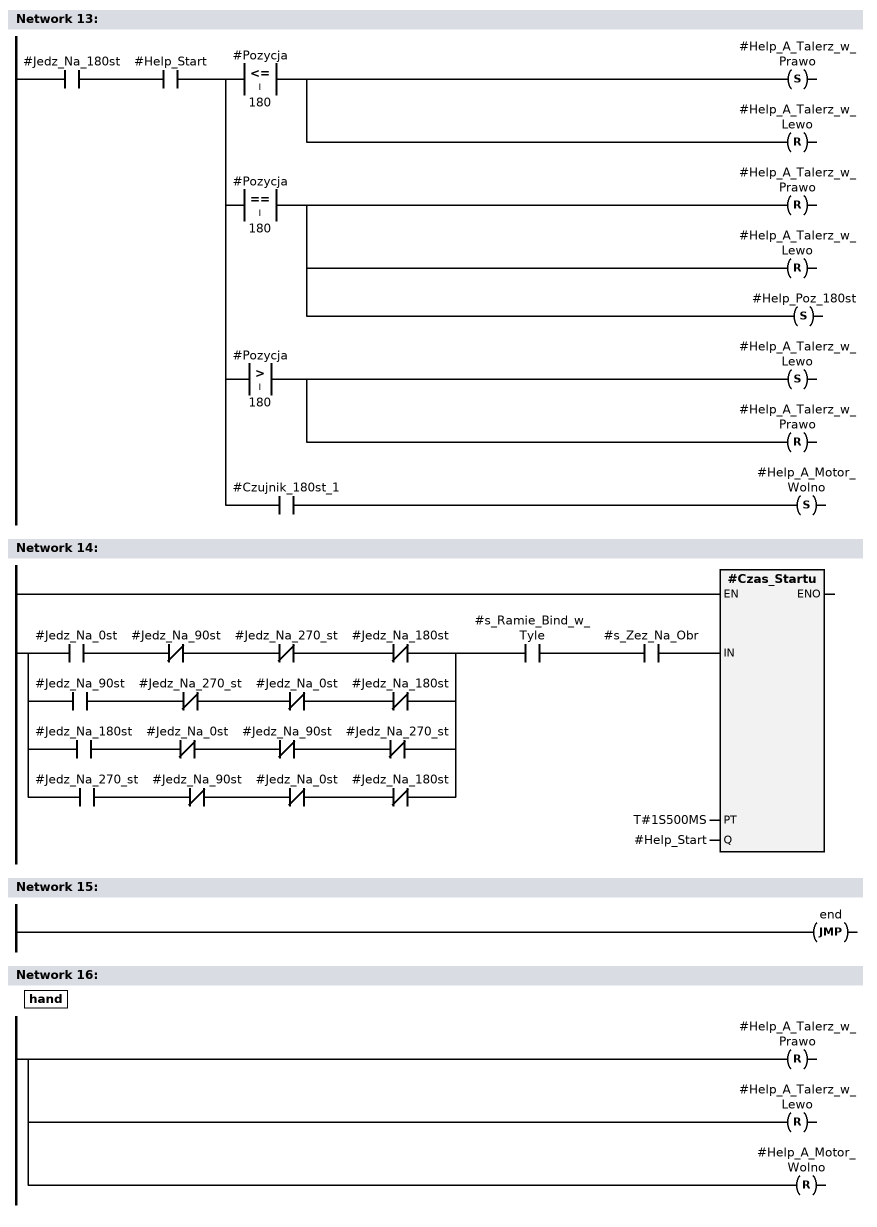
NETWORK
TITLE =
//Jazda na 180 st od strony lewej i od strony prawej. Gdy najazd od strony lewej 
//najpierw jest hamowanie talerza nastepnie zatrzymanie. Gdy najazd od strony 
//prawej nastepuje miniecie czujnika nastepnie zatrzymanie i cofniecie
//
//
      A     #Jedz_Na_180st;
      A     #Help_Start;
      =     L 1.0;
      A     L 1.0;
      A(;
      L     #Pozycja;
      L     180;
      <=I;
      );
      S     #Help_A_Talerz_w_Prawo;
      R     #Help_A_Talerz_w_Lewo;
      A     L 1.0;
      A(;
      L     #Pozycja;
      L     180;
      ==I;
      );
      R     #Help_A_Talerz_w_Prawo;
      R     #Help_A_Talerz_w_Lewo;
      S     #Help_Poz_180st;
      A     L 1.0;
      A(;
      L     #Pozycja;
      L     180;
      >I;
      );
      S     #Help_A_Talerz_w_Lewo;
      R     #Help_A_Talerz_w_Prawo;
      A     L 1.0;
      A     #Czujnik_180st_1;
      S     #Help_A_Motor_Wolno;
NETWORK
TITLE =
//Opoznienie startu po wydaniu rozkazu
      A(;
      A     #Jedz_Na_0st;
      AN    #Jedz_Na_90st;
      AN    #Jedz_Na_270_st;
      AN    #Jedz_Na_180st;
      O;
      A     #Jedz_Na_90st;
      AN    #Jedz_Na_270_st;
      AN    #Jedz_Na_0st;
      AN    #Jedz_Na_180st;
      O;
      A     #Jedz_Na_180st;
      AN    #Jedz_Na_0st;
      AN    #Jedz_Na_90st;
      AN    #Jedz_Na_270_st;
      O;
      A     #Jedz_Na_270_st;
      AN    #Jedz_Na_90st;
      AN    #Jedz_Na_0st;
      AN    #Jedz_Na_180st;
      );
      A     #s_Ramie_Bind_w_Tyle;
      A     #s_Zez_Na_Obr;
      =     L 1.0;
      BLD   103;
      CALL  #Czas_Startu (
           IN                       := L 1.0,
           PT                       := T#1S500MS,
           Q                        := #Help_Start);
      NOP   0;
NETWORK
TITLE =
//Koniec tryby automatycznego
//
      JU    end;
NETWORK
TITLE =
//tryb reczny
hand: NOP   0;
      SET;
      R     #Help_A_Talerz_w_Prawo;
      R     #Help_A_Talerz_w_Lewo;
      R     #Help_A_Motor_Wolno;
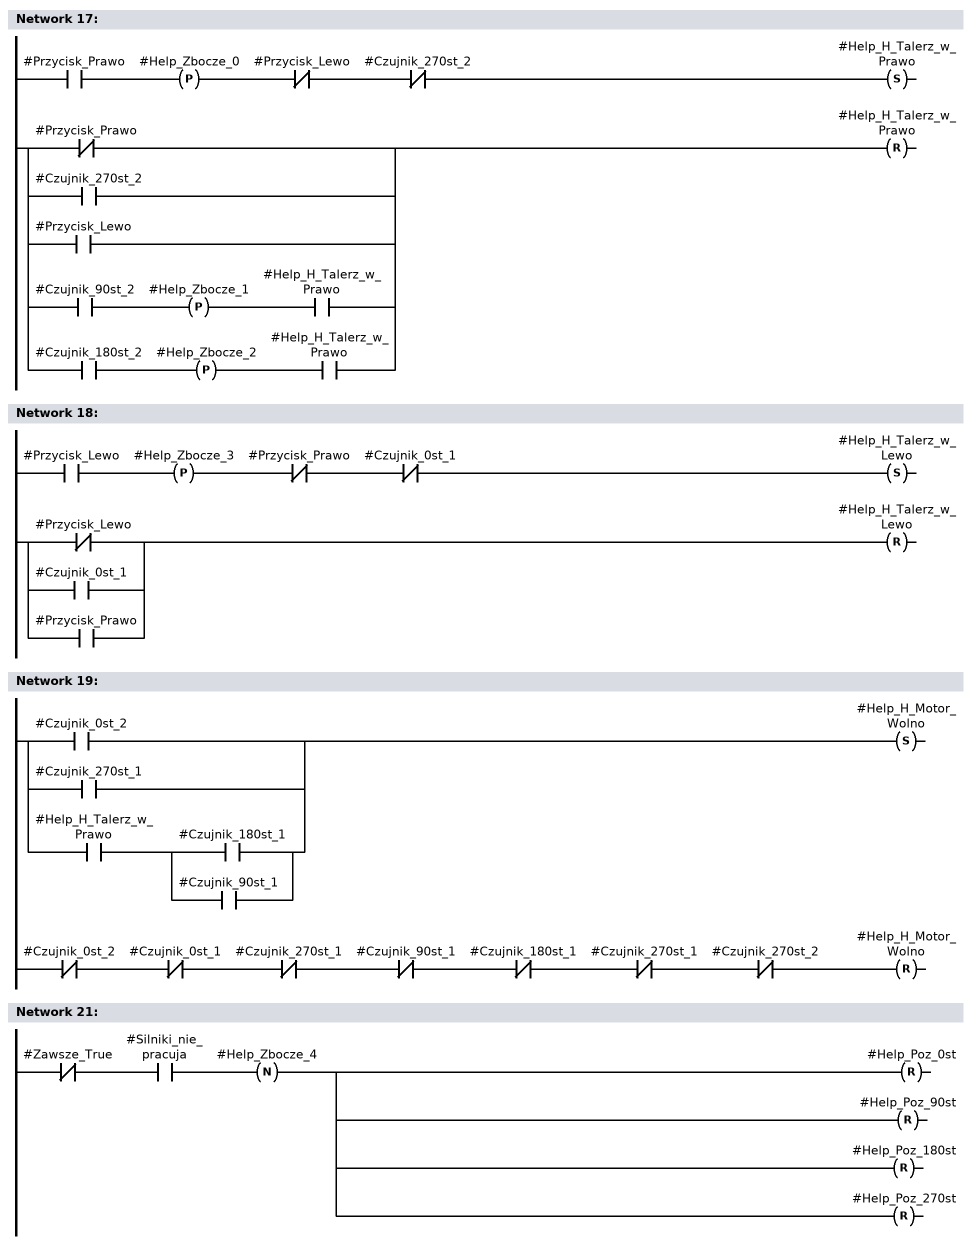
NETWORK
TITLE =
//Ruch talerza w prawo i zatrzymywanie sie na pozycji
//
      A     #Przycisk_Prawo;
      FP    #Help_Zbocze_0;
      AN    #Przycisk_Lewo;
      AN    #Czujnik_270st_2;
      S     #Help_H_Talerz_w_Prawo;
      A(;
      ON    #Przycisk_Prawo;
      O     #Czujnik_270st_2;
      O     #Przycisk_Lewo;
      O(;
      A     #Czujnik_90st_2;
      FP    #Help_Zbocze_1;
      A     #Help_H_Talerz_w_Prawo;
      );
      O(;
      A     #Czujnik_180st_2;
      FP    #Help_Zbocze_2;
      A     #Help_H_Talerz_w_Prawo;
      );
      );
      R     #Help_H_Talerz_w_Prawo;
      NOP   0;
NETWORK
TITLE =
//Ruch talerza w lewo. Zatrzymanie tylko na skrajnych pozycjach
//
      A     #Przycisk_Lewo;
      FP    #Help_Zbocze_3;
      AN    #Przycisk_Prawo;
      AN    #Czujnik_0st_1;
      S     #Help_H_Talerz_w_Lewo;
      A(;
      ON    #Przycisk_Lewo;
      O     #Czujnik_0st_1;
      O     #Przycisk_Prawo;
      );
      R     #Help_H_Talerz_w_Lewo;
      NOP   0;
NETWORK
TITLE =
//Zwolnienie predkosci gdy jazda w trybie recznym 
      A(;
      O     #Czujnik_0st_2;
      O     #Czujnik_270st_1;
      O;
      A     #Help_H_Talerz_w_Prawo;
      A(;
      O     #Czujnik_180st_1;
      O     #Czujnik_90st_1;
      );
      );
      S     #Help_H_Motor_Wolno;
      AN    #Czujnik_0st_2;
      AN    #Czujnik_0st_1;
      AN    #Czujnik_270st_1;
      AN    #Czujnik_90st_1;
      AN    #Czujnik_180st_1;
      AN    #Czujnik_270st_1;
      AN    #Czujnik_270st_2;
      R     #Help_H_Motor_Wolno;
      NOP   0;
NETWORK
TITLE =
end:  NOP   0;
NETWORK
TITLE =
//resetowanie pozycji gdy silniki rusza.
//Rozkaz kasowania wyciety
      AN    #Zawsze_True;
      A     #Silniki_nie_pracuja;
      FN    #Help_Zbocze_4;
      R     #Help_Poz_0st;
      R     #Help_Poz_90st;
      R     #Help_Poz_180st;
      R     #Help_Poz_270st;
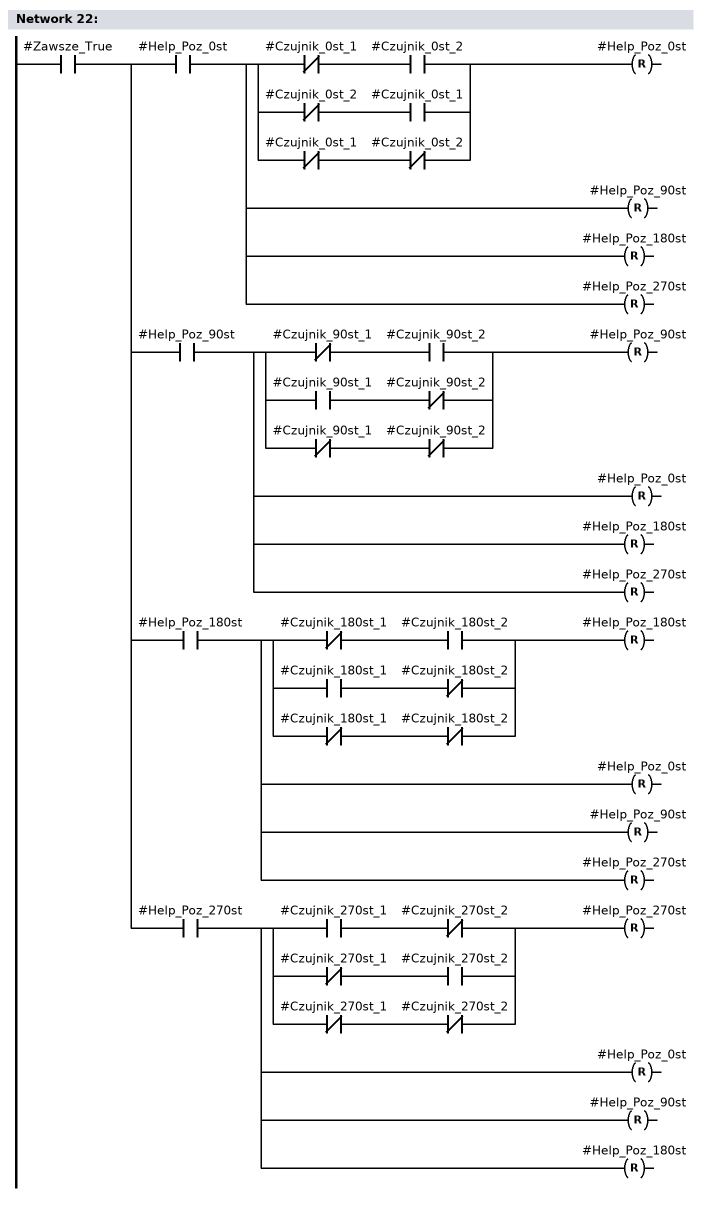
NETWORK
TITLE =
//The can be only one.
      A     #Zawsze_True;
      =     L 1.0;
      A     L 1.0;
      A     #Help_Poz_0st;
      =     L 1.1;
      A     L 1.1;
      A(;
      AN    #Czujnik_0st_1;
      A     #Czujnik_0st_2;
      O;
      AN    #Czujnik_0st_2;
      A     #Czujnik_0st_1;
      O;
      AN    #Czujnik_0st_1;
      AN    #Czujnik_0st_2;
      );
      R     #Help_Poz_0st;
      A     L 1.1;
      BLD   102;
      R     #Help_Poz_90st;
      A     L 1.1;
      BLD   102;
      R     #Help_Poz_180st;
      A     L 1.1;
      BLD   102;
      R     #Help_Poz_270st;
      A     L 1.0;
      A     #Help_Poz_90st;
      =     L 1.1;
      A     L 1.1;
      A(;
      AN    #Czujnik_90st_1;
      A     #Czujnik_90st_2;
      O;
      A     #Czujnik_90st_1;
      AN    #Czujnik_90st_2;
      O;
      AN    #Czujnik_90st_1;
      AN    #Czujnik_90st_2;
      );
      R     #Help_Poz_90st;
      A     L 1.1;
      BLD   102;
      R     #Help_Poz_0st;
      A     L 1.1;
      BLD   102;
      R     #Help_Poz_180st;
      A     L 1.1;
      BLD   102;
      R     #Help_Poz_270st;
      A     L 1.0;
      A     #Help_Poz_180st;
      =     L 1.1;
      A     L 1.1;
      A(;
      AN    #Czujnik_180st_1;
      A     #Czujnik_180st_2;
      O;
      A     #Czujnik_180st_1;
      AN    #Czujnik_180st_2;
      O;
      AN    #Czujnik_180st_1;
      AN    #Czujnik_180st_2;
      );
      R     #Help_Poz_180st;
      A     L 1.1;
      BLD   102;
      R     #Help_Poz_0st;
      A     L 1.1;
      BLD   102;
      R     #Help_Poz_90st;
      A     L 1.1;
      BLD   102;
      R     #Help_Poz_270st;
      A     L 1.0;
      A     #Help_Poz_270st;
      =     L 1.1;
      A     L 1.1;
      A(;
      A     #Czujnik_270st_1;
      AN    #Czujnik_270st_2;
      O;
      AN    #Czujnik_270st_1;
      A     #Czujnik_270st_2;
      O;
      AN    #Czujnik_270st_1;
      AN    #Czujnik_270st_2;
      );
      R     #Help_Poz_270st;
      A     L 1.1;
      BLD   102;
      R     #Help_Poz_0st;
      A     L 1.1;
      BLD   102;
      R     #Help_Poz_90st;
      A     L 1.1;
      BLD   102;
      R     #Help_Poz_180st;
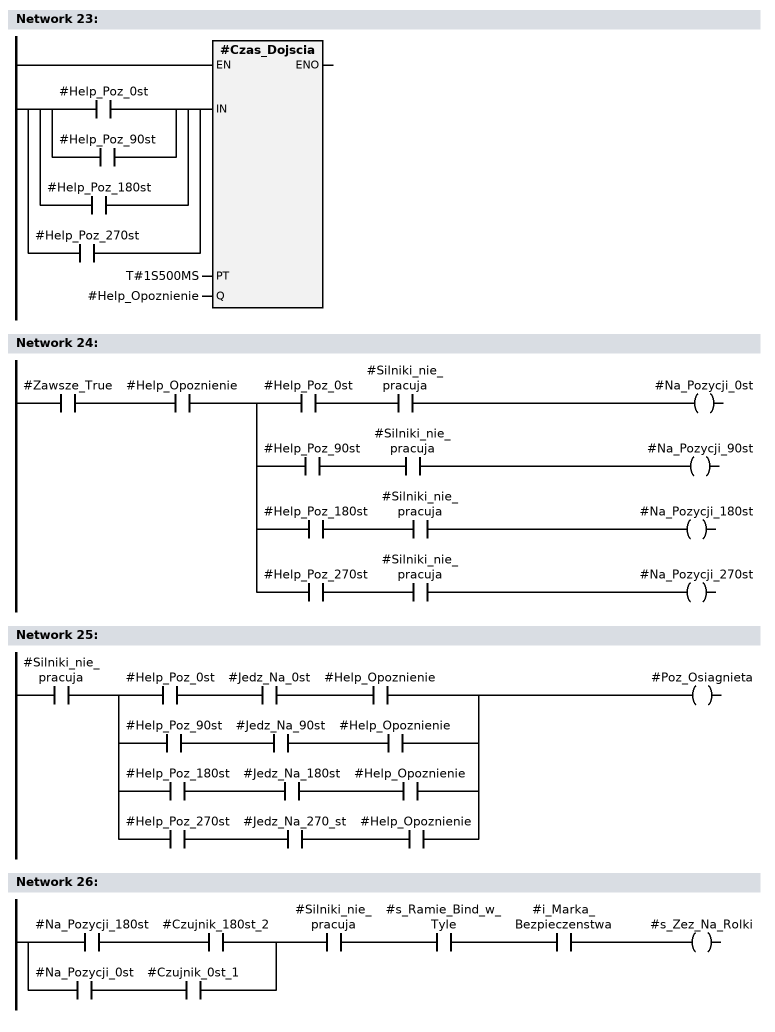
NETWORK
TITLE =
//Opoznienie potwierdzenia pozycji
      A(;
      O     #Help_Poz_0st;
      O     #Help_Poz_90st;
      O     #Help_Poz_180st;
      O     #Help_Poz_270st;
      );
      =     L 1.0;
      BLD   103;
      CALL  #Czas_Dojscia (
           IN                       := L 1.0,
           PT                       := T#1S500MS,
           Q                        := #Help_Opoznienie);
      NOP   0;
NETWORK
TITLE =
//przypisanie pozycji
//
      A     #Zawsze_True;
      A     #Help_Opoznienie;
      =     L 1.0;
      A     L 1.0;
      A     #Help_Poz_0st;
      A     #Silniki_nie_pracuja;
      =     #Na_Pozycji_0st;
      A     L 1.0;
      A     #Help_Poz_90st;
      A     #Silniki_nie_pracuja;
      =     #Na_Pozycji_90st;
      A     L 1.0;
      A     #Help_Poz_180st;
      A     #Silniki_nie_pracuja;
      =     #Na_Pozycji_180st;
      A     L 1.0;
      A     #Help_Poz_270st;
      A     #Silniki_nie_pracuja;
      =     #Na_Pozycji_270st;
NETWORK
TITLE =
//Potwierdzenie osiagniecia pozycji
      A     #Silniki_nie_pracuja;
      A(;
      A     #Help_Poz_0st;
      A     #Jedz_Na_0st;
      A     #Help_Opoznienie;
      O;
      A     #Help_Poz_90st;
      A     #Jedz_Na_90st;
      A     #Help_Opoznienie;
      O;
      A     #Help_Poz_180st;
      A     #Jedz_Na_180st;
      A     #Help_Opoznienie;
      O;
      A     #Help_Poz_270st;
      A     #Jedz_Na_270_st;
      A     #Help_Opoznienie;
      );
      =     #Poz_Osiagnieta;
NETWORK
TITLE =
//Warunek odblokowanch rolek
      A(;
      A     #Na_Pozycji_180st;
      A     #Czujnik_180st_2;
      O;
      A     #Na_Pozycji_0st;
      A     #Czujnik_0st_1;
      );
      A     #Silniki_nie_pracuja;
      A     #s_Ramie_Bind_w_Tyle;
      A     #i_Marka_Bezpieczenstwa;
      =     #s_Zez_Na_Rolki;
